(* CoDeSys 2.3 export: OSCAT311.TXT *)
(* Libraries: Standard.lib 4.10.05 11:14:46 *)

(* Global variable list: Constants *)
VAR_GLOBAL CONSTANT
	STRING_LENGTH : INT := 250;
	NETWORK_BUFFER_LONG_SIZE : UINT := 3999;
	NETWORK_BUFFER_SHORT_SIZE : UINT := 1459;
END_VAR




(* revisionhistory
hm 3. mar. 2007
	extended accuracy of pi2
	renamed T0 to Tk for better compatibility with other libraries
	renamed C t0 c0 for better compatibility

hm	2. may. 2007
	added RU universal gas constant

hm	1. oct. 2007
	added setup parameter STEP7

hm 31. oct. 2007
	added PN

hm	6. mar. 2008
	added setup Parameter EXTENDED_ASCII

hm	28. Mar. 2008
	added setup parameter STRING_LENGTH

hm	7. apr. 2008
	Deleted unused setup parameter Step7

hm	19. apr. 2008
	added setup parameter NETWORK_BUFFER_SIZE

hm	27. apr. 2008
	added PI05 and PI025

hm	18. may. 2008
	added charname lists
	renamed E to E1

hm	30. jun. 2008
	reduced size of string constants to 253 to avoid problems with target aixia DCUF

hm	21. sep. 2008
	added section language setup
	added section location setup

hm	20. oct. 2008
	changed to structured constants

hm	16. nov. 2008
	moved structured constants to global vars for compatibility reasons

hm	13. nov. 2009
	added network_buffer_short_size
	renamed network_buffer_long_size
	changed string length to 250
*)

(* Global variable list: Globale_Variablen *)
VAR_GLOBAL
	MATH : CONSTANTS_MATH;
	PHYS : CONSTANTS_PHYS;
	LANGUAGE : CONSTANTS_LANGUAGE;
	SETUP : CONSTANTS_SETUP;
	LOCATION : CONSTANTS_LOCATION;
END_VAR

(* Data type *)
TYPE CALENDAR :
STRUCT
	UTC : DT;						(* world time UTC *)
	LDT : DT;						(* local time *)
	LDATE : DATE;				(* local date *)
	LTOD : TOD;					(* local time of day *)
	YEAR : INT;					(* year of LDATE *)
	MONTH : INT;					(* month of LDATE *)
	DAY : INT;						(* day of LDATE *)
	WEEKDAY : INT;				(* weekday of LDATE *)
	OFFSET : INT;					(* Time Zone Offset for Local time in minutes *)
	DST_EN : BOOL;				(* daylight savings time enable *)
	DST_ON : BOOL;				(* true when daylight savings time os on *)
	NAME : STRING(5);			(* name of time zone *)
	LOCATION : INT;				(* location number pls see location setup *)
	LONGITUDE : REAL;			(* longitude of current location *)
	LATITUDE : REAL;			(* latitude of current location *)
	SUN_RISE : TOD;				(* sun_rise for current location *)
	SUN_SET : TOD;				(* sun_set for current location *)
	SUN_MIDDAY : TOD;			(* worldtime when sun stands at south position *)
	SUN_HEIGTH : REAL	;		(* suns heigth at midday, south position *)
	SUN_HOR : REAL;			(* sun angle horizontal 0 = north in degrees *)
	SUN_VER : REAL;			(* sun angle vertical above horizon in degrees *)
	NIGHT : BOOL;				(* true between sun_set and sun_rise *)
	HOLIDAY : BOOL;				(* true when holiday *)
	HOLY_NAME : STRING(30);	(* name of holiday *)
	WORK_WEEK : INT;			(* current work week *)
END_STRUCT
END_TYPE

(* revision history
hm	21. nov. 2008	rev 1.0
	original version

hm	8. feb. 2009	rev 1.1
	added sun position data

hm	10. mar. 2009	rev 1.2
	added work_week, sun_midday, sun_heigth
*)

(* Data type *)
TYPE COMPLEX :
STRUCT
	re : REAL;
	im : REAL;
END_STRUCT
END_TYPE


(* revision history
hm	18. oct. 2008
	original version

*)

(* Data type *)
TYPE CONSTANTS_LANGUAGE :
STRUCT
	(* Language Setup *)
	DEFAULT : INT := 1; (* 1=english, 2=german 3=french *)
	LMAX : INT := 3;
	WEEKDAYS : ARRAY[1..3, 1..7] OF STRING(10) :=	'Monday', 'Tuesday', 'Wednesday', 'Thursday', 'Friday', 'Saturday', 'Sunday',
													'Montag', 'Dienstag', 'Mittwoch', 'Donnerstag', 'Freitag', 'Samstag', 'Sonntag',
													'Lundi', 'Mardi', 'Mercredi', 'Jeudi', 'Vendredi', 'Samedi', 'Dimanche';
	WEEKDAYS2 : ARRAY[1..3, 1..7] OF STRING(2) :=	'Mo', 'Tu', 'We', 'Th', 'Fr', 'Sa', 'Su',
													'Mo', 'Di', 'Mi', 'Do', 'Fr', 'Sa', 'So',
													'Lu', 'Ma', 'Me', 'Je', 'Ve', 'Sa', 'Di';
	MONTHS : ARRAY[1..3, 1..12] OF STRING(10) :=	'January', 'February', 'March', 'April', 'May', 'June', 'July', 'August', 'September', 'October', 'November', 'December',
													'Januar', 'Februar', 'März', 'April', 'Mai', 'Juni', 'Juli', 'August', 'September', 'Oktober', 'November', 'Dezember',
													'Janvier', 'Février', 'mars', 'Avril', 'Mai', 'Juin', 'Juillet', 'Août', 'Septembre', 'Octobre', 'Novembre', 'Decembre';
	MONTHS3 : ARRAY[1..3, 1..12] OF STRING(3) :=	'Jan', 'Feb', 'Mar', 'Apr', 'May', 'Jun', 'Jul', 'Aug', 'Sep', 'Oct', 'Nov', 'Dec',
													'Jan', 'Feb', 'Mrz', 'Apr', 'Mai', 'Jun', 'Jul', 'Aug', 'Sep', 'Okt', 'Nov', 'Dez',
													'Jan', 'Fev', 'Mar', 'Avr', 'Mai', 'Jun', 'Jul', 'Aou', 'Sep', 'Oct', 'Nov', 'Dec';
	DIRS : ARRAY[1..3,0..15] OF STRING(3) :=		'N', 'NNE', 'NE', 'ENE', 'E', 'ESE', 'SE', 'SSE', 'S', 'SSW', 'SW', 'WSW', 'W', 'WNW', 'NW', 'NNW',
													'N', 'NNO', 'NO', 'ONO', 'O', 'OSO', 'SO', 'SSO', 'S', 'SSW', 'SW', 'WSW', 'W', 'WNW', 'NW', 'NNW',
													'N', 'NNO', 'NO', 'ONO', 'O', 'OSO', 'SO', 'SSO', 'S', 'SSW', 'SW', 'WSW', 'W', 'WNW', 'NW', 'NNW';
END_STRUCT
END_TYPE

(* revision history
hm	19. oct. 2008	rev 1.0
	original version

hm	22. oct. 2008	rev 1.1
	added directions DIRS

hm	23. dec. 2008	rev 1.2
	added french language

*)

(* Data type *)
TYPE CONSTANTS_LOCATION :
STRUCT
	(* location setup *)
	DEFAULT : INT := 1; (* 1=germany, 2=austria 3=france *)
	LMAX : INT := 3;

	(*	if month = 0 then F_day is the offset in days from easter
		used :0 = NOT used, 1 = used, -1..-7 menas the weekday before the specified DATE example -3 means wednesday before 23.11
	*)
	HOLIDAY : ARRAY[1..3, 0..29] OF HOLIDAY_DATA := (name := 'Neujahr', day := 1, month := 1, use := 1),
													(name := 'Heilig Drei Könige', day := 6, month := 1, use := 1),
													(name := 'Karfreitag', day := -2, month := 0, use := 1),
													(name := 'Ostersonntag', day := 0, month := 0, use := 1),
													(name := 'Ostermontag', day := 1, month := 0, use := 1),
													(name := 'Tag der Arbeit', day := 1, month := 5, use := 1),
													(name := 'Christi Himmelfahrt', day := 39, month := 0, use := 1),
													(name := 'Pfingstsonntag', day := 49, month := 0, use := 1),
													(name := 'Pfingstmontag', day := 50, month := 0, use := 1),
													(name := 'Fronleichnam', day := 60, month := 0, use := 1),
													(name := 'Augsburger Friedensfest', day := 8, month := 8, use := 0),
													(name := 'Maria Himmelfahrt', day := 15, month := 8, use := 1),
													(name := 'Tag der Deutschen Einheit', day := 3, month := 10, use := 1),
													(name := 'Reformationstag', day := 31, month := 10, use := 0),
													(name := 'Allerheiligen', day := 1, month := 11, use := 1),
													(name := 'Buss und Bettag', day := 23, month := 11, use := 0),
													(name := '1. Weihnachtstag', day := 25, month := 12, use := 1),
													(name := '2. Weihnachtstag', day := 26, month := 12, use := 1),
													(),
													(),
													(),
													(),
													(),
													(),
													(),
													(),
													(),
													(),
													(),
													(),
													(* the next 30 lines are for austrian holidays *)
													(name := 'Neujahr', day := 1, month := 1, use := 1),
													(name := 'Heilig Drei Könige', day := 6, month := 1, use := 1),
													(name := 'Karfreitag', day := -2, month := 0, use := 1),
													(name := 'Ostersonntag', day := 0, month := 0, use := 1),
													(name := 'Ostermontag', day := 1, month := 0, use := 1),
													(name := '', day := 1, month := 5, use := 0),
													(name := 'Christi Himmelfahrt', day := 39, month := 0, use := 1),
													(name := 'Pfingstsonntag', day := 49, month := 0, use := 1),
													(name := 'Pfingstmontag', day := 50, month := 0, use := 1),
													(name := 'Fronleichnam', day := 60, month := 0, use := 1),
													(name := '', day := 8, month := 8, use := 0),
													(name := 'Maria Himmelfahrt', day := 15, month := 8, use := 1),
													(name := '', day := 3, month := 10, use := 0),
													(name := '', day := 31, month := 10, use := 0),
													(name := 'Allerheiligen', day := 1, month := 11, use := 1),
													(name := 'Maria Empfängnis', day := 8, month := 12, use := 1),
													(name := '1. Weihnachtstag', day := 25, month := 12, use := 1),
													(name := '2. Weihnachtstag', day := 26, month := 12, use := 1),
													(),
													(),
													(),
													(),
													(),
													(),
													(),
													(),
													(),
													(),
													(),
													(),
													(* the next 30 lines are for french holidays *)
													(name := 'Nouvel an', day := 1, month := 1, use := 1),
													(name := 'St Valentin', day := 14, month := 2, use := 0),
													(name := 'Vendredi Saint (alsace)', day := -2, month := 0, use := 0),
													(name := 'Dimanche de pâques', day := 0, month := 0, use := 1),
													(name := 'Lundi de pâques', day := 1, month := 0, use := 1),
													(name := 'Jeudi de Ascension', day := 39, month := 0, use := 1),
													(name := 'dimanche de Pentecôte ', day := 49, month := 0, use := 1),
													(name := 'jeudi de la Trinité', day := 60, month := 0, use := 0),
													(name := 'Fête du travail', day := 1, month := 5, use := 1),
													(name := 'Victoire 1945 ', day := 8, month := 5, use := 1),
													(name := 'Prise de La bastille', day := 14, month := 7, use := 1),
													(name := '15 Août 1944', day := 15, month := 8, use := 1),
													(name := 'Halloween', day := 31, month := 10, use := 0),
													(name := 'Armistice 1918', day := 11, month := 11, use := 1),
													(name := 'Noël', day := 25, month := 12, use := 1),
													(name := 'Saint Étienne (alsace)', day := 26, month := 12, use := 0),
													(name := 'Fête de la musique', day := 21, month := 6, use := 0),
													(),
													(),
													(),
													(),
													(),
													(),
													(),
													(),
													(),
													(),
													(),
													(),
													();

END_STRUCT
END_TYPE


(* revision history
hm	20. oct. 2008	rev 1.0
	original version

hm	23. dec. 2008	rev 1.1
	added french holidays
*)

(* Data type *)
TYPE CONSTANTS_MATH :
STRUCT
	PI : REAL := 	3.14159265358979323846264338327950288;	(* Kreiszahl PI *)
	PI2 : REAL := 	6.28318530717958647692528676655900576;	(* PI * 2 *)
	PI4 : REAL :=  12.56637061435917295385057353311801152;	(* PI * 4 *)
	PI05 : REAL :=  1.5707963267949;						(* PI / 2 *)
	PI025 : REAL := 0.785398163397448;						(* PI / 4 *)
	PI_INV : REAL := 0.318309886183791;						(* 1 / PI *)
	E : REAL := 	2.71828182845904523536028747135266249;	(* Eulersche Konstante e *)
	E_INV : REAL := 0.367879441171442;						(* 1 / e *)
	SQ2 : REAL :=	1.4142135623731;						(* Wurzel von 2 *)
END_STRUCT
END_TYPE



(* revision history
hm	26.10.2008	rev 1.0
	original version

*)

(* Data type *)
TYPE CONSTANTS_PHYS :
STRUCT
	C : REAL := 299792458.0;				(* Lichtgeschwindigkeit in m/s *)
	E : REAL := 1.60217653E-19;				(* elementarladung in Colomb = A * s *)
	G : REAL := 9.80665; 						(* Erdbeschleunigung in m / s² *)
	T0 : REAL := -273.15;						(* absoluter Nullpunkt in °C *)
	RU : REAL := 8.314472; 					(* Universelle Gaskonstante in J / (mol · K) *)
	PN : REAL := 101325.0;					(* NormalDruck in Pa *)
END_STRUCT
END_TYPE



(* revision history
hm	18.10.2008	rev 1.0
	original version

hm	13. mar. 2009	rev 1.1
	real constants updated to new systax using dot

*)

(* Data type *)
TYPE CONSTANTS_SETUP :
STRUCT
	(* setup Parameters *)
	EXTENDED_ASCII : BOOL := TRUE;
	CHARNAMES : ARRAY[1..4] OF STRING(253) := ';"&quot;&&amp;<&lt;>&gt;€&euro; &nbsp;¡&iexcl;¢&cent;£&pound;¤&curren;¥&yen;¦&brvbar;§&sect;¨&uml;©&copy;ª&ordf;«&laquo;¬&not;­&shy;®&reg;¯&macr;°&deg;±&plusmn;²&sup2;³&sup3;´&acute;µ&micro;¶&para;·&middot;¸&cedil;¹&sup1;º&ordm;»&raquo;¼&frac14;Û&Ucirc;',
		';¾&frac34;¿&iquest;À&Agrave;Á&Aacute;Â&Acirc;Ã&Atilde;Ä&Auml;Å&Aring;Æ&AElig;Ç&Ccedil;È&Egrave;É&Eacute;Ê&Ecirc;Ë&Euml;Ì&Igrave;Í&Iacute;Î&Icirc;Ï&Iuml;Ð&ETH;Ñ&Ntilde;Ò&Ograve;Ó&Oacute;Ô&Ocirc;Õ&Otilde;Ö&Ouml;×&times;Ø&Oslash;Ù&Ugrave;Ú&Uacute;½&frac12;',
		';Ü&Uuml;Ý&Yacute;Þ&THORN;ß&szlig;à&agrave;á&aacute;â&acirc;ã&atilde;ä&auml;å&aring;æ&aelig;ç&ccedil;è&egrave;é&eacute;ê&ecirc;ë&euml;ì&igrave;í&iacute;î&icirc;ï&iuml;ð&eth;ñ&ntilde;ò&ograve;ó&oacute;ô&ocirc;õ&otilde;ö&ouml;÷&divide;ø&oslash;ù&ugrave;',
		';ú&uacute;û&ucirc;ü&uuml;ý&yacute;þ&thorn;ÿ&yuml;';
	MTH_OFS : ARRAY[1..12] OF INT := 0,31,59,90,120,151,181,212,243,273,304,334;
	DECADES : ARRAY[0..8] OF REAL := 1,10,100,1000,10000,10000,100000,1000000,10000000;
END_STRUCT
END_TYPE

(* revision history
hm	24.10.2008	rev 1.0
	original version

*)

(* Data type *)
TYPE ESR_DATA :
STRUCT
	TYP : BYTE;
	ADRESS : STRING(10);
	DS : DT;
	TS : TIME;
	DATA : ARRAY[0..7] OF BYTE;
END_STRUCT
END_TYPE


(* revision history
hm	18. oct. 2008
	original version

*)

(* Data type *)
TYPE HOLIDAY_DATA :
STRUCT
	NAME : STRING(30);
	DAY : SINT;
	MONTH : SINT;
	USE : SINT;
END_STRUCT
END_TYPE


(* revision history
hm	18. oct. 2008
	original version

*)

(* Data type *)
TYPE NETWORK_BUFFER :
STRUCT
	SIZE : UINT;
	BUFFER : NW_BUF_LONG;
END_STRUCT
END_TYPE


(* revision history
hm	18. oct. 2008
	original version

hm 13. nov. 2009
	use constant network_buffer_long_size

*)

(* Data type *)
TYPE NETWORK_BUFFER_SHORT :
STRUCT
	SIZE : UINT;
	BUFFER : NW_BUF_SHORT;
END_STRUCT
END_TYPE


(* revision history
hm 13. nov. 2009
	original version

*)

(* Data type *)
TYPE
	NW_BUF_LONG  : ARRAY[0..NETWORK_BUFFER_LONG_SIZE] OF BYTE;
END_TYPE

(* Data type *)
TYPE
	NW_BUF_SHORT : ARRAY[0..NETWORK_BUFFER_SHORT_SIZE] OF BYTE;
END_TYPE

(* Data type *)
TYPE REAL2 :
STRUCT
	R1 : REAL;	(* small value *)
	RX : REAL;	(* big value *)
END_STRUCT
END_TYPE


(* revision history
hm	18. oct. 2008
	original version

*)

(* Data type *)
TYPE SDT :
STRUCT
	YEAR : INT;
	MONTH : INT;
	DAY : INT;
	WEEKDAY : INT;
	HOUR : INT;
	MINUTE : INT;
	SECOND : INT;
	MS : INT;
END_STRUCT
END_TYPE


(* revision history
hm	18. oct. 2008
	original version

*)

(* Data type *)
TYPE TIMER_EVENT :
STRUCT
	TYP : BYTE;
	CHANNEL : BYTE;
	DAY : BYTE;
	START : TOD;
	DURATION : TIME;
	LAND : BYTE;
	LOR : BYTE;
	LAST : DWORD;
END_STRUCT
END_TYPE


(* revision history
hm	18. oct. 2008
	original version

*)

(* Data type *)
TYPE URL :
STRUCT
	PROTOCOL : STRING(10);
	USER : STRING(20);
	PASSWORD : STRING(20);
	DOMAIN : STRING(80);
	PORT : WORD;
	PATH : STRING(80);
	QUERY : STRING(40);
	ANCHOR : STRING(40);
END_STRUCT
END_TYPE


(* revision history
hm	18. oct. 2008
	original version

*)

(* Data type *)
TYPE VECTOR_3 :
STRUCT
	X : REAL;
	Y : REAL;
	Z : REAL;
END_STRUCT
END_TYPE


(* revision history
hm	18. oct. 2008
	original version

*)

(* POU PLC_PRG, CFC *)
PROGRAM PLC_PRG
VAR
END_VAR
_CFC_ (* Continuous Function Chart, elements in execution order *)
_END_CFC_
END_PROGRAM

(* POU Buffer Management/_BUFFER_CLEAR, ST *)
FUNCTION _BUFFER_CLEAR : BOOL
VAR_INPUT
	PT : POINTER TO BYTE;
	SIZE : UINT;
END_VAR
VAR
	ptw : POINTER TO DWORD;
	temp: DWORD;
	end, end32 : DWORD;
END_VAR


(*
version 1.2	31. oct. 2008
programmer 	hugo
tested by	oscat

this function will initialize a given array of byte with 0.
the function needs to be called:	_buffer_clear(adr("array"),sizeof("array"));
this function will manipulate a given array.
the function manipulates the original array, it rerturnes true when finished.
because this function works with pointers its very time efficient and it needs no extra memory.

*)
(* this routine uses 32 bit access to gain speed *)
(* first access bytes till pointer is aligned for 32 bit access *)
temp := pt;
end := temp + UINT_TO_DWORD(size);
end32 := end - 3;
WHILE (pt < end) AND ((temp AND 16#00000003) > 0) DO
	pt^ := 0;
	pt := pt + 1;
	temp := temp + 1;
END_WHILE;
(* pointer is aligned, now copy 32 bits at a time *)
ptw := pt;
WHILE ptw < end32 DO (* *)
	ptw^ := 0;
	ptw := ptw + 4;
END_WHILE;
(* copy the remaining bytes in byte mode *)
pt := ptw;
WHILE pt < end DO
	pt^ := 0;
	pt := pt + 1;
END_WHILE;

_BUFFER_CLEAR := TRUE;

(* revision History
hm 	5. mar. 2008	rev 1.0
	original version

hm	16. mar. 2008	rev 1.1
	added type conversion to avoid warnings under codesys 30
	chaged type of input size to uint
	deleted unused variable i

hm	31. oct. 2008	rev 1.2
	corrected an error while routine would write outside of arrays

*)
END_FUNCTION

(* POU Buffer Management/_BUFFER_INIT, ST *)
FUNCTION _BUFFER_INIT : BOOL
VAR_INPUT
	PT : POINTER TO BYTE;
	SIZE : UINT;
	INIT : BYTE;
END_VAR
VAR
	ptw : POINTER TO DWORD;
	temp : DWORD;
	end, end32 : DWORD;
END_VAR


(*
version 1.2	31. oct. 2008
programmer 	hugo
tested by	oscat

this function will initialize a given array of byte with init.
the function needs to be called:	_buffer_init(adr("array"),sizeof("array"),init);
this function will manipulate a given array.
the function manipulates the original array, it rerturnes true when finished.
because this function works with pointers its very time efficient and it needs no extra memory.

*)
(* this routine uses 32 bit access to gain speed *)
(* first access bytes till pointer is aligned for 32 bit access *)
temp := pt;
end := temp + UINT_TO_DWORD(size);
end32 := end - 3;
WHILE (pt < end) AND ((temp AND 16#00000003) > 0) DO
	pt^ := init;
	pt := pt + 1;
	temp := temp + 1;
END_WHILE;
(* pointer is aligned, now copy 32 bits at a time *)
ptw := pt;
temp := SHL(BYTE_TO_DWORD(init),24) OR SHL(BYTE_TO_DWORD(init),16) OR SHL(BYTE_TO_DWORD(init),8) OR BYTE_TO_DWORD(init);
WHILE ptw < end32 DO
	ptw^ := temp;
	ptw := ptw + 4;
END_WHILE;
(* copy the remaining bytes in byte mode *)
pt := ptw;
WHILE pt < end DO
	pt^ := init;
	pt := pt + 1;
END_WHILE;

_BUFFER_INIT := TRUE;

(* revision History
hm 	5. mar. 2008	rev 1.0
	original version

hm	16. mar. 2008	rev 1.1
	added type conversion to avoid warnings under codesys 3.0
	chaged type of input size to uint.

hm	31. oct. 2008	rev 1.2
	corrected an error while routine would write outside of arrays

*)
END_FUNCTION

(* POU Buffer Management/_BUFFER_INSERT, ST *)
FUNCTION _BUFFER_INSERT : BOOL
VAR_INPUT
	STR : STRING(STRING_LENGTH);
	POS : INT;
	PT : POINTER TO ARRAY[0..32767] OF BYTE;
	SIZE : UINT;
END_VAR
VAR
	end : INT;
	lx: INT;
	i: INT;
END_VAR


(*
version 1.4	12. nov. 2009
programmer 	hugo
tested by		oscat

this function will initialize a given array of byte with init.
the function needs to be called:	_buffer_init(adr("array"),sizeof("array"),init);
this function will manipulate a given array.
the function manipulates the original array, it rerturnes true when finished.
because this function works with pointers its very time efficient and it needs no extra memory.

*)
lx := LEN(str);
end := pos + lx;
(* first move the upper part of the buffer to make space for the string *)
FOR i := UINT_TO_INT(size) - 1 TO end BY -1 DO
	pt^[i] := pt^[i-lx];
END_FOR;
(* copy the string *)
_BUFFER_INSERT := _STRING_TO_BUFFER(str, pos, PT, size);


(* revision History
hm 	9. mar. 2008	rev 1.0
	original version

hm	16. mar. 2008	rev 1.1
	changed type of input size to uint

hm	13. may. 2008	rev 1.2
	changed type of pointer to array[1..32767]
	changed size of string to STRING_LENGTH

hm	23. mar. 2009	rev 1.3
	avoid writing to input pos

hm	12. nov. 2009	rev 1.4
	code optimized

*)
END_FUNCTION

(* POU Buffer Management/_STRING_TO_BUFFER, ST *)
FUNCTION _STRING_TO_BUFFER : BOOL
VAR_INPUT
	STR : STRING(STRING_LENGTH);
	POS : INT;
	PT : POINTER TO ARRAY[0..32767] OF BYTE;
	SIZE : UINT;
END_VAR
VAR
	ps : POINTER TO BYTE;
	i: INT;
	end: INT;
END_VAR


(*
version 1.3	12. nov. 2009
programmer 	hugo
tested by		oscat

this function will copy a string into an array of byte starting at position pos.
the function needs to be called:	_String_To_buffer(str, pos, adr("array"),sizeof("array"));
this function will manipulate the array directly in memory and returns true when finished.
because this function works with pointers its very time efficient and it needs no extra memory.

*)
ps := ADR(str);
end := MIN(pos + LEN(str), UINT_TO_INT(size));
IF end > 0 THEN end := end -1; END_IF;
FOR i := pos TO end DO
	pt^[i] := ps^;
	ps := ps + 1;
END_FOR;

_STRING_TO_BUFFER := TRUE;

(* revision History

hm 	5. mar. 2008	rev 1.0
	original version

hm	16. mar. 2008	rev 1.1
	changed type of input size to uint

hm	13. may. 2008	rev 1.2
	changed type of pointer to array[1..32767]
	changed size of string to STRING_LENGTH

hm	12. nov. 2009	rev 1.3
	limit end to size - 1

*)
END_FUNCTION

(* POU Buffer Management/BUFFER_COMP, ST *)
FUNCTION BUFFER_COMP : INT
VAR_INPUT
	PT1 : POINTER TO ARRAY[0..32767] OF BYTE;
	SIZE1 : INT;
	PT2 : POINTER TO ARRAY[0..32767] OF BYTE;
	SIZE2 : INT;
	START : INT;
END_VAR
VAR
	i, j, end : INT;
	firstbyte: BYTE;
END_VAR

(*
version 1.1	12. nov. 2009
programmer 	hugo
tested by	oscat


 
*)
(* search for first character match *)
IF size2 <= size1 THEN
	end := size1 - size2;
	firstbyte := PT2^[0];
	FOR i := START TO end DO
		IF PT1^[i] = firstbyte THEN
			(* first character matches, now compare rest of array *)
			j := 1;
			WHILE j < size2 DO
				IF pt2^[j] <> pt1^[j+i] THEN EXIT; END_IF;
				j := j + 1;
			END_WHILE;
			(* when J > size2 a match was found return the position i in buffer1 *)
			IF j = size2 THEN
				BUFFER_COMP := i;
				RETURN;
			END_IF;
		END_IF;
	END_FOR;
END_IF;
BUFFER_COMP := -1;


(*
hm 14. nov. 2008	rev 1.0
	original version

hm	12. nov. 2009	rev 1.1
	performance increase

*)
END_FUNCTION

(* POU Buffer Management/BUFFER_SEARCH, ST *)
FUNCTION BUFFER_SEARCH : INT
VAR_INPUT
	PT : POINTER TO ARRAY[0..32767] OF BYTE;
	SIZE : UINT;
	STR : STRING(STRING_LENGTH);
	POS : UINT;
	IGN : BYTE;
END_VAR
VAR
	ps : POINTER TO ARRAY[0..255] OF BYTE;
	i: INT;
	end: INT;
	k: INT;
	lx: INT;
END_VAR


(*
version 1.3	12. nov. 2009
programmer 	hugo
tested by	oscat

this function will search for a string STR in an array of byte starting at position pos.
the function needs to be called:	buffer_search(adr("array"),sizeof("array"), STR, POS, IGN);
because this function works with pointers its very time efficient and it needs no extra memory.
The function returns the position of the first character of the string in the array if found.
a 0 is returned if the string is not found in the array.
The parameter IGN specifies a wildcard character in the search string.

*)
ps := ADR(str);
lx := LEN(str);
end := MIN(UINT_TO_INT(size) - lx, UINT_TO_INT(size - 1));
lx := lx - 1;
FOR i := UINT_TO_INT(pos) TO end DO
	FOR k := 0 TO lx DO
		IF (ps^[k] <> ign) AND (ps^[k] <> pt^[i+k]) THEN EXIT; END_IF;
	END_FOR;
	IF k > lx THEN
		BUFFER_SEARCH := i;
		RETURN;
	END_IF;
END_FOR;
BUFFER_SEARCH := 0;


(* revision History

hm 5. mar. 2008	rev 1.0
	original version

hm	16. mar. 2008	rev 1.1
	chaged type of input size to uint

hm	13. may. 2008	rev 1.2
	changed type of pointer to array[1..32767]
	changed size of string to STRING_LENGTH

hm	12. nov. 2009	rev 1.3
	limit end to array size

*)
END_FUNCTION

(* POU Buffer Management/BUFFER_TO_STRING, ST *)
FUNCTION BUFFER_TO_STRING : STRING(STRING_LENGTH)
VAR_INPUT
	PT : POINTER TO ARRAY[0..32767] OF BYTE;
	SIZE : UINT;
	START : UINT;
	STOP : UINT;
END_VAR
VAR
	ps : POINTER TO BYTE;
	i : UINT;
	stp: UINT;
	sta: UINT;
END_VAR


(*
version 1.5	12. nov. 2009
programmer 	hugo
tested by		oscat

this function will retrieve a string from an array of byte starting at position start and stop at position stop.
the function needs to be called:	buffer_TO_String(adr("array"),sizeof("array"), start, stop);
because this function works with pointers its very time efficient and it needs no extra memory.

*)
ps := ADR(BUFFER_TO_STRING);
IF size = 0 THEN RETURN; END_IF;
sta := MIN(start, size -1);
stp := MIN(stop, size -1);

(* check for maximum string_length *)
IF UINT_TO_INT(stp - sta + 1) >= STRING_LENGTH THEN
	stp := sta + INT_TO_UINT(STRING_LENGTH) - 1;
END_IF;

FOR i := sta TO stp DO
	ps^ := pt^[i];
	ps := ps + 1;
END_FOR;

(* terminate the string *)

ps^ := 0;



(* revision History
hm 	5. mar. 2008	rev 1.0
	original version

hm	16. mar. 2008	rev 1.1
	changed type of input size to uint

hm	13. may. 2008	rev 1.2
	changed type of pointer to array[0..32767]
	changed size of string to STRING_LENGTH

hm	12. jun. 2008	rev 1.3
	check for pointer overrun
	change input start and stop to uint
	added type conversions to avoid warnings under codesys 3.0

hm	23. mar. 2009	rev 1.4
	avoid writing to input stop

hm	12. nov. 2009 rev 1.5
	limit start and stop to size -1

*)
END_FUNCTION

(* POU Building/actuators/ACTUATOR_2P, ST *)
FUNCTION_BLOCK ACTUATOR_2P
VAR_INPUT
	IN : BYTE;
	TEST : BOOL;
	ARE : BOOL := TRUE;
END_VAR
VAR_IN_OUT
	ARX : BOOL;
END_VAR
VAR_INPUT CONSTANT
	CYCLE_TIME : TIME;
	SENS : BYTE;
	SELF_ACT_TIME : TIME;
	SELF_ACT_PULSE : TIME;
	SELF_ACT_CYCLES : INT := 1;
END_VAR
VAR_OUTPUT
	OUT : BOOL;
	ARO : BOOL;
END_VAR
VAR
	timer : AUTORUN;
	pwgen : GEN_PULSE;
END_VAR


(*
version 2.1	24. jan. 2009
programmer 	hugo
tested by		oscat

this is an intelligent actuator interface for any 2point actuator like coil drive.
the 2Point actuator can only switch on/off and therefore the input must be converted to on/off cycles.
the interface can be programmed with double click on the symbol.
in addition a self_act_time and self_act_cycles ca be programmed to switch n times on/off every self_act_time to avoid a valve to freeze.
the input value must be between 0 and 255. with the setup variable sens one can specify what must be the minimum input to turn the valve on at all.
at the same time an input > 255-sens will turn the valve on at all times.


*)
(* run the autorun timer *)
timer(trun := SELF_ACT_PULSE * (2 * SELF_ACT_CYCLES), toff := SELF_ACT_TIME, Test := TEST, ARE := ARE, arx := ARX);
ARO := timer.ARO;

(* run the pulse width generator *)
IF aro THEN
	pwgen(PTL := SELF_ACT_PULSE, PTH := SELF_ACT_PULSE);
	out := pwgen.Q;
ELSIF in < sens THEN
	out := FALSE;
ELSIF in > BYTE#255 - sens THEN
	out := TRUE;
ELSE
	pwgen.PTH := (CYCLE_TIME * BAND_B(IN,SENS)) / 255;
	pwgen.PTL := CYCLE_TIME - pwgen.PTH;
	pwgen();
	out := pwgen.Q;
END_IF;



(* revision history
hm	7.10.2006 		rev 1.1
	changed error pos could not reach 1 or 0 under certain conditions due to error in code.
	changed on and off in force and force_in for better usability.

hm	17.1.2007		rev 1.2
	deleted unused variable time_overflow

hm	15.9.2007		rev 1.3
	replaced time() with T_PLC_MS for compatibility and performance reasons

hm	19. 11 2007		rev 1.4
	replaced left over statement time() with tx

hm	27. 12. 2007	REV 1.5
	CHANGED CODE FOR BETTER PERFORMANCE

hm	21. oct. 2008	rev 1.6
	code optimized

hm	23. nov. 2008	rev 2.0
	new code using library modules

hm	24. jan. 2009	rev 2.1
	deleted unused var inb
*)
END_FUNCTION_BLOCK

(* POU Engineering/measurements/CYCLE_TIME, ST *)
FUNCTION_BLOCK CYCLE_TIME
VAR_INPUT
	RST : BOOL;
END_VAR
VAR_OUTPUT
	ct_min : TIME;
	ct_max : TIME;
	ct_last : TIME;
	systime : TIME;
	sysdays : INT;
	cycles : DWORD;
END_VAR
VAR
	last_cycle : TIME;
	tx: TIME;
	init: BOOL;
END_VAR


(*
	version 1.2	16 sep 2007
	programmer 	hugo
	tested BY		hans

this function block measures the cycle time and displays the last, min and max cycle time of the current task.
the resolution is 1ms.
the cycles output is a dword counter which counts the cycles.
a rst pulse on the input will reset all data.


*)
tx := DWORD_TO_TIME(T_PLC_MS()) - last_cycle;
IF rst THEN
	ct_min := t#10h;
	ct_max := t#0ms;
	cycles := 0;
ELSIF last_cycle > t#0s THEN
	IF tx < ct_min THEN ct_min := tx;
	ELSIF tx > ct_max THEN ct_max := tx;
	END_IF;
	ct_last := tx;
ELSIF ct_min = t#0s THEN
	ct_min := t#0s - t#1ms;
END_IF;
IF init THEN
	systime := systime + tx;
		IF systime >= t#1d THEN
			systime := systime - t#1d;
			sysdays := sysdays + 1;
		END_IF;
END_IF;
init := TRUE;
last_cycle := last_cycle + tx;
cycles := cycles + 1;

(*	revision history
hm 12.12.2006		rev 1.1
	added cycles output, a dword cycle counter.
hm 10.3.2007			rev 1.2
	changed initialization of ct_min to t#10h for compatibility with siemens s7

hm	16.9.2007		rev 1.2
	changed Time() in T_PLC_MS() for compatibility resons

*)
END_FUNCTION_BLOCK

(* POU Engineering/measurements/T_PLC_MS, ST *)
FUNCTION T_PLC_MS : DWORD
VAR CONSTANT
	debug : BOOL := 0;
	N : INT := 0;
	offset : DWORD := 0;
END_VAR
VAR
	tx : TIME;
END_VAR

(*
version 1.2	16. nov 2008
programmer 	hugo
tested by	oscat

T_PLC_MS reads the internal PLC timer and return the time, it has the advantage to be able to set a debug mode 
and speed up the counter to test the plc timer overrun which occurs every 50 days respectively 25 days at siemens S7
this routine also allows to correct the behavior of s7 where the internal plc counter will not count all 32 bits.

*)
tx := TIME();
T_PLC_MS := TIME_TO_DWORD(Tx);
(* hier muss die korrektur für step7 stattfinden
plctime muss den vollen wertebereich von time ausnutzen:
wenn bei step7 time -24tage bis plus 24 tage ist dann muss der timer auch beim überlauf auf -24tage springen 
und auf keinen fall auf 0 !!!!
für siemens muss ein weiterer fb im main eingebunden werden der sicherstellt das alle 32 bits durchgezählt werden.
es kann nur ein fb sein den er muss sich das oberste (32te) bit merken.
oder etwa spring s7 bei überlauf auf -24 tage????? dann wäre keine korrektur nötig.
*)
IF debug THEN
	T_PLC_MS := (SHL(T_PLC_MS,N) OR SHL(DWORD#1,N)-1) + OFFSET;
END_IF;

(* revision history
hm	14.9.2007	rev 1.0
	original version

hm	12. nov 2007	rev 1.1
	added temporaray variable tx because some compilers could not handle time() as an argument

hm	16. nov. 2008	rev 1.2
	initialized constants with 0 for compatibility reasons
*)
END_FUNCTION

(* POU Engineering/signal processing/OFFSET, ST *)
FUNCTION OFFSET : REAL
VAR_INPUT
	X : REAL;
	O1, O2, O3, O4 : BOOL;
	D : BOOL;
END_VAR
VAR_INPUT CONSTANT
	Offset_1 : REAL;
	Offset_2 : REAL;
	Offset_3 : REAL;
	Offset_4 : REAL;
	default : REAL;
END_VAR

(*
version 1.0	12 jan 2007
programmer 	oscat
tested by	oscat

The Function offset adds offsets to an analog signal depending on digital inputs.
all selected offsets are added at the same time.
with the input D a default value instead of the input X can be used.

*) 
IF D THEN OFFSET := default; ELSE OFFSET := X; END_IF;
IF O1 THEN OFFSET := OFFSET + offset_1; END_IF;
IF O2 THEN OFFSET := OFFSET + offset_2; END_IF;
IF O3 THEN OFFSET := OFFSET + offset_3; END_IF;
IF O4 THEN OFFSET := OFFSET + offset_4; END_IF;



(* revision history
hm	12. jan 2007
	original version


*)
END_FUNCTION

(* POU Building/actuators/AUTORUN, ST *)
FUNCTION_BLOCK AUTORUN
VAR_INPUT
	IN : BOOL;
	TEST : BOOL;
	ARE : BOOL := TRUE;
END_VAR
VAR_IN_OUT
	ARX : BOOL;
END_VAR
VAR_INPUT CONSTANT
	TRUN : TIME;
	TOFF : TIME;
END_VAR
VAR_OUTPUT
	OUT : BOOL;
	ARO : BOOL;
END_VAR
VAR
	timer : _RMP_B;
	val : BYTE;
END_VAR



(*
version 1.0	20. nov 2008
programmer 	hugo
tested by	oscat




*)
(* run the integrator when T_off > T#0s *)
IF TOFF > T#0s THEN
	timer(DIR:= OUT, TR := SEL(OUT, TOFF, TRUN), RMP := val);
ELSE
	val := 255;
END_IF;


(* when timer = 0 or test then initiate autorun until timer reaches 255 *)
IF (NOT ARX AND ARE AND val = 0) OR TEST THEN
	val := 0;
	ARO := TRUE;
	ARX := TRUE;
ELSIF val = 255 AND ARO THEN
	ARO := FALSE;
	ARX := FALSE;
END_IF;

(* output is true when autorun ARO is true or in = TRUE *)
out := IN OR ARO;



(* revision history
hm 20. nov. 2008	rev 1.0
	original version

*)
END_FUNCTION_BLOCK

(* POU Engineering/signal generators/_RMP_B, ST *)
FUNCTION_BLOCK _RMP_B
VAR_INPUT
	DIR : BOOL;  (* true = up *)
	E : BOOL := TRUE;
	TR : TIME;
END_VAR
VAR_IN_OUT
	RMP : BYTE;
END_VAR
VAR
	tx, tl : DWORD;
	step : INT;
	init: BOOL;
	last_dir: BOOL;
END_VAR


(*
version 1.1	20. nov. 2008
programmer 	hugo
tested by	oscat


_RMP_B generates a ramp on an external var of type byte
tr is the total ramp time, E is an enable and dir the direction of the ramp

*)
tx := T_PLC_MS();
IF E AND init THEN
	(* we need to set tl = tx when direction changes *)
	IF dir XOR last_dir THEN
	 tl := tx;
	 last_dir := dir;
	END_IF;
	(* check_elapsed time and calculate only if necessary *)
	IF tr > t#0s THEN
		step := DWORD_TO_INT(SHL(tx-tl, 8) / TIME_TO_DWORD(TR));
	ELSE
		step := 255;
	END_IF;
	IF step > 0 THEN
		(* perform the step on the ramp *)
		tl := tx;
		(* calculate the step response *)
		IF NOT dir THEN step := - step; END_IF;
		rmp := INT_TO_BYTE(LIMIT(0, BYTE_TO_INT(rmp) + step, 255));
	END_IF;
ELSE
	tl := tx;
	init := TRUE;
END_IF;


(* revison history
hm	22. oct. 2008	rev 1.0
	original version

hm	20. nov. 2008	rev 1.1
	set default for E to be TRUE
	added init

*)
END_FUNCTION_BLOCK

(* POU Engineering/signal generators/GEN_PULSE, ST *)
FUNCTION_BLOCK GEN_PULSE
VAR_INPUT
	ENQ : BOOL := TRUE;
	PTH : TIME;
	PTL : TIME;
END_VAR
VAR_OUTPUT
	Q : BOOL;
END_VAR
VAR
	tx: TIME;
	tn: TIME;
	init: BOOL;
END_VAR

(*
version 1.3	13. nov. 2009
programmer 	hugo
tested by		oscat

GEN_PULSE uses the internal sps timer to generate a continuous output waveform with programmable high and low time.
the accuracy of gen_pulse is depending on the system timer.
when time is 0 the high and low times are exactly one cycle.
ENQ = TRUE will start and ENQ = FALSE will stop the generator.

*)
(* read system timer *)
IF enq THEN
	tx := DWORD_TO_TIME(T_PLC_MS());
	IF NOT init THEN init := TRUE; tn := tx; END_IF;
	IF tx >= tn THEN
		Q := NOT Q;
		tn := tn + SEL(Q,PTL,PTH);
	END_IF;
ELSE
	Q := FALSE;
	init := FALSE;
END_IF;



(* revision history
hm	29. jun. 2008	rev 1.0
	original version

hm	23. nov. 2008	rev 1.1
	set default for enq to be true

hm	18. jul. 2009	rev 1.2
	improved performance

hm	13. nov. 2009	rev 1.3
	corrected error

*)
END_FUNCTION_BLOCK

(* POU Engineering/control/BAND_B, ST *)
FUNCTION BAND_B : BYTE
VAR_INPUT
	X : BYTE;
	B : BYTE;
END_VAR



(*
version 1.0	21. Nov. 2008
programmer 	hugo
tested by	oscat

BAND_B will limit X to B <= X <= 255-B. while X < B the resulkt will be 0 and while X > 255-B the output will be 255
otherwise the result = X.

*)
IF X < B THEN
	BAND_B := 0;
ELSIF X > BYTE#255-B THEN
	BAND_B := 255;
ELSE
	BAND_B := X;
END_IF;



(* revision history
hm	21. nov. 2008	rev 1.0
	original version

*)
END_FUNCTION

(* POU Building/actuators/ACTUATOR_3P, ST *)
FUNCTION_BLOCK ACTUATOR_3P
VAR_INPUT
	in : REAL;
	force : BOOL;
	on : BOOL;
	end_pos : BOOL;
	diag : BOOL;
END_VAR
VAR_INPUT CONSTANT
	min_ontime : TIME := t#10s;
	min_offtime : TIME := t#10s;
	max_runtime : TIME := t#60s;
	auto_diag_time : TIME := t#10d;
	cal_runtime : TIME := t#600s;
	switch_available: BOOL;
END_VAR
VAR_OUTPUT
	out1 : BOOL;
	out2 : BOOL;
	pos : REAL;
	busy : BOOL;
	error : BOOL;
END_VAR
VAR
	val: REAL;
	tx : TIME;
	last_diag: TIME;
	last : TIME;
	runtime_1 : TIME;
	runtime_2 : TIME;
	state : INT;
	rout: FT_RMP;
	end : R_TRIG;
	cal_timer: TIME;
	Tn: TIME;
END_VAR


(*
version 1.3	 15 sep 2007
programmer 	hugo
tested by	oscat

actuator_3P is an interface for a 3 point actuator.
a 3P actuator is a motor with 2 directions that drives a valve or flap. the position of the valve or flap is controlled by runtime of the motor foreward or backward.
the available inputs are:
in is a real value which specifies the position of the actuator, 0 = 0% and 1 = 100% any value <0 or > 1 is limited to 0 or 1.
a force input must be low for normal operation and if switched high, the motor can only be controlled for 0% or 100% positions with the on input.
an and pos input is available for a end_pos switch, this switch indicates the valve or flap to be at either 0% or 100%
a diag input can at any time start a diag cycle which turns the motor towards the 0% position, then measures the runtime to 100% and then the runtime to 0%
these runtimes are stored and used for absolute positioning of the motor during normal operation.
a setup constand "auto_diag_time can be used to specify how often the actuator repeates this auto_diag cycla automatically.
at power on a cycle is perfomed automatically.
a 0 for this value means auto diag is never performed.

the outputs ar out1 and out2 for up and down direction of the motor. to avoid flickering the output can be programmed for min_ontime and min_offtime.
a pos outout indicates the absulute position of the actuator during operation and a busy output indicates the actuator is busy.
a error output is initiated when the specified max_runtime is reached by any direction during debug.
also when the up and down direction differs by more then 10% the error output is set.

for absolute positioning accuracy the actuator has a setup variable "cal_runtime" if this is set the actuator measures the total runtime of the motors and when this 
cal_runtime is exceeded it resets the actuator to 0% position and sets the output again to assure absolute accuracy.

autodiag and calibration can be shut off by setting the appropriate values to 0.
a switch_available setup variable specifies if end_pos switches are available.

*)
(* setup *)
Tn := DWORD_TO_TIME(T_PLC_MS());
tx := Tn - last;
end(clk := end_pos);

(* init only when first started *)
IF state = 0 THEN
	runtime_1 := max_runtime;
	runtime_2 := max_runtime;
	state := 1;
	rout(KR := 1000 / TIME_TO_REAL(runtime_1), KF := 1000 / TIME_TO_REAL(runtime_1) );
	tx := t#0s;
	last := Tn;
	last_diag := last;
END_IF;

(* check for end_sw and stop if reached *)
IF switch_available AND out1 AND end.Q THEN
	(* upper limit has been reached *)
	out1 := 0;
	rout(rmp := 0, in := 1);
	rout.Rmp := 1;
ELSIF switch_available AND out2 AND end.Q THEN
	(* lower limit has been reached *)
	out2 := 0;
	rout(rmp := 0, in := 0);
	rout.Rmp := 1;
END_IF;

(* check for min_offtime and min_ontime and return if it has not elapsed *)
IF NOT busy AND tx < min_offtime THEN
	RETURN;
ELSIF busy AND tx < min_ontime THEN
	RETURN;

(* check for last diag cycle and start diag if auto_diag_time has elapsed *)
ELSIF (tn - last_diag > auto_diag_time AND state > 10 AND auto_diag_time > t#0s) OR (diag AND state >= 10) THEN state := 1;

(* check if force pin is high *)
ELSIF force THEN state := 10;

(* check if calibration is necessary *)
ELSIF cal_timer > cal_runtime AND state = 99 AND cal_runtime > t#0s THEN state := 20;
END_IF;

(* state machine for operation *)
CASE state OF

1 :	(* diagnostic start *)
	(* all data is reset and out2 is turned on to make sure we start from top position *)
	last_diag := tn;
	diag := 0;
	state := 2;
	pos := 0;
	busy := 1;
	last := tn;
	out1 := 0;
	out2 := 1;
	RETURN;

2:	(* wait for max_runtime or end_pos to be reached *)
	IF tx < max_runtime AND NOT end.Q THEN RETURN; END_IF;
	state := 3;
	last := tn;
	out1 := 1;
	out2 := 0;
	RETURN;

3: 	(* measure runtime_2 *)
	IF tx < max_runtime AND NOT end.Q THEN RETURN; END_IF;
	state := 4;
	runtime_1 := tx;
	last := tn;
	out1 := 0;
	out2 := 1;
	RETURN;

4:	(* measure runtime_1 *)
	IF tx < max_runtime AND NOT end.Q THEN RETURN; END_IF;
	state := 99;
	runtime_2 := tx;
	last := tn;
	out2 := 0;
	busy := 0;
	(* reset the output ramp generator to the 0% position as the valve is after diags *)
	rout(rmp := 0, in := 0);
	rout.Rmp := 1;
	cal_timer := t#0s;
	IF DIFFER(TIME_TO_REAL(runtime_1), TIME_TO_REAL(runtime_2), TIME_TO_REAL(max_runtime) * 0.1) THEN error := TRUE;
	ELSIF runtime_1 > MULTIME(max_runtime, 0.9) AND switch_available THEN error := TRUE;
	ELSIF runtime_2 > MULTIME(max_runtime, 0.9) AND switch_available THEN error := TRUE;
	END_IF;
	RETURN;

10: (* force pin is active, outputs are forced on or off by the on pin *)
	IF on AND NOT out2 THEN val := 1;
	ELSIF NOT on AND NOT out1 THEN val := 0;
	END_IF;
	IF NOT force THEN state := 99; END_IF;

20 : (* calibrate to allow for correction of positioning error addig up *)
	cal_timer := t#0s;
	state := 21;
	pos := 0;
	busy := 1;
	last := tn;
	out1 := 0;
	out2 := 1;
	RETURN;

21:	(* after end_sw or max_runtime we can be sure to have reached the 0% position *)
	IF tx < max_runtime AND NOT end.Q THEN RETURN; END_IF;
	state := 99;
	out2 := 0;
	busy := 0;
	last := tn;
	rout(rmp := 0, in := 0);
	rout.Rmp := 1;
	RETURN;

99: (* normal operation *)
	(* only if input changes for an equivalent of min_ontime then change the output *)
	(* if there is a directional change then wait until last step is finished *)
	IF in < TIME_TO_REAL(min_ontime)/TIME_TO_REAL(max_runtime)/2 THEN val := 0;
	ELSIF in > 1 - TIME_TO_REAL(min_ontime)/TIME_TO_REAL(max_runtime)/2 THEN val := 1;
	ELSIF differ(LIMIT(0,in,1), val, TIME_TO_REAL(min_ontime) / TIME_TO_REAL(max_runtime)) OR in = 0 OR in = 1 THEN
		IF in < val AND NOT out1 THEN val := in;
		ELSIF in > val AND NOT out2 THEN val := in;
		END_IF;
	END_IF;

END_CASE;

(* output ramp generator *)
rout(in := val);
out1 := rout.busy AND rout.UD;
out2 := rout.busy AND NOT rout.UD;
pos := rout.out;

(* set the busy output and if busy goes low, then set the last time in order to check for min_offtime *)
IF NOT busy AND rout.busy THEN
	last := tn;
ELSIF busy AND NOT rout.busy THEN
	cal_timer := cal_timer + tx;
	last := tn;
END_IF;
busy := rout.busy;



(* revision history

19.10.2006	rev 1.1
	added security checks for end_switch to avoid overrun of the end_switch, hans

23.1.2007		rev 1.2
	deleted unused variables force_on and force_off

15.9.2007	hm	rev 1.3
	replaced Time() with T_PLC_MS for compatibility and performance reasons

*)
END_FUNCTION_BLOCK

(* POU Mathematical/functions/FT_RMP, ST *)
FUNCTION_BLOCK FT_RMP
VAR_INPUT
	Rmp : BOOL := TRUE;
	in : REAL;
	KR : REAL;
	KF : REAL;
END_VAR
VAR_OUTPUT
	out : REAL;
	busy : BOOL;
	UD : BOOL;
END_VAR
VAR
	tx: TIME;
	last: TIME;
	init: BOOL;
END_VAR

(*
	version 1.4	25 jan 2008
	programmer 	oscat
	tested BY		oscat

this ramp function follows an input signal with a linear ramp up or down, the up or down speed can be set with KF and KR.
a K factor of 1 means 1 unit per second on the output. K factors can only be positive and not negative.
a busy output signals the ramp is running or busy false means the in value is present on the output.
a rmp input false means the output follows the input dierctly while a rmp = true means the output follows the input with a ramp.
a updn output signal the directon of the ramp (up or down).

*)
(* read system time *)
tx := DWORD_TO_TIME(T_PLC_MS()) - last;

IF NOT init THEN
	init := TRUE;
	last := tx;
	tx := t#0s;
	out := in;
END_IF;
IF NOT rmp THEN
	out := in;
	busy := FALSE;
ELSIF out > in THEN
	(* ramp down *)
	out := out - TIME_TO_REAL(tx) * 0.001 * KF;
	out := MAX(in, out);
ELSIF out < in THEN
	(* ramp up *)
	out := out + TIME_TO_REAL(tx) * 0.001 * KR;
	out := MIN(in, out);
END_IF;

(* set busy and dir flags *)
IF out < in THEN
	busy := TRUE;
	ud := TRUE;
ELSIF out > in THEN
	busy := TRUE;
	ud := FALSE;
ELSE
	busy := FALSE;
END_IF;
last := last + tx;


(* revision history:

hm 8.10.2006			rev 1.1
	added ud output

hm 12. feb 2007		rev 1.2
	added init variable and corrected a possible startup problem

hm	17. sep 2007	rev 1.3
	replaced time() with t_plc_ms() for compatibility reasons

hm	25. jan 2008	rev 1.4
	performance improvements
	allow KR and KF to be 0
*)
END_FUNCTION_BLOCK

(* POU Mathematical/DIFFER, ST *)
FUNCTION DIFFER : BOOL
VAR_INPUT
	in1 : REAL;
	in2 : REAL;
	X : REAL;
END_VAR


(*
version 1.1	16 mar 2008
programmer 	hugo
tested by		tobias

this function checks if in1 differs more then x from in2
the output is true if abs(in1-in2) > X

*)
DIFFER := ABS(in1 - in2) > X;

(* revision history
hm		8. oct 2006		rev 1.0
	original version

hm		16. mar 2008	rev 1.1
	improverd code for performance

*)
END_FUNCTION

(* POU Time&Date/MULTIME, ST *)
FUNCTION MULTIME : TIME
VAR_INPUT
	t : TIME;
	M : REAL;
END_VAR


(*
version 1.1	14 mar 2008
programmer 	hugo
tested by		tobias

multiplies a time by a real number and returns a time
*)
MULTIME := DWORD_TO_TIME(REAL_TO_DWORD(DWORD_TO_REAL(TIME_TO_DWORD(t))*M));

(* revision history
hm		2. oct 2006	rev 1.0
	original version

hm		14. mar 2008	rev 1.1
	rounded the result after the last digit

*)
END_FUNCTION

(* POU Building/actuators/ACTUATOR_A, ST *)
FUNCTION_BLOCK ACTUATOR_A
VAR_INPUT
	I1 : BYTE;
	IS : BOOL;
	I2 : BYTE;
	RV : BOOL;
	DX : BOOL;
END_VAR
VAR_INPUT CONSTANT
	RUNTIME : TIME;
	SELF_ACT_TIME : TIME;
	OUT_MIN : WORD;
	OUT_MAX : WORD;
END_VAR
VAR_OUTPUT
	Y : WORD;
END_VAR
VAR
	timer : CYCLE_4;
	dx_edge: BOOL;
END_VAR


(*
version 1.0 8. nov. 2008	
programmer 	hugo
tested by	oscat

ACTUATOR_A drives any valve or similar with 0 - 255 continuous control input.
 
*)
(* run the system timer, if self_act_time = t#0s then state is set to 0 *)
timer(T0 := RUNTIME, T1 := RUNTIME, T3 := SELF_ACT_TIME, sl := DX AND NOT dx_edge, sx := 0, S0 := SELF_ACT_TIME > t#0s);
dx_edge := dx;

CASE timer.STATE OF
	0: 	(* self act min value *)
		Y := OUT_MIN;
	1:	(* self_act max value *)
		Y := OUT_MAX;
	3:	(* normal operation *)
		IF rv THEN
			Y := OUT_MAX - (OUT_MAX - OUT_MIN) * SEL(IS, I1, I2) / 255;
		ELSE
			Y := (OUT_MAX - OUT_MIN) * SEL(IS, I1, I2) / 255 + OUT_MIN;
		END_IF;
END_CASE;




(*
hm 	8. nov. 2008	rev 1.0
	original version

*)
END_FUNCTION_BLOCK

(* POU Logic/generators/CYCLE_4, ST *)
FUNCTION_BLOCK CYCLE_4
VAR_INPUT
	E : BOOL := TRUE;
	T0, T1, T2, T3 : TIME;
	S0 : BOOL;
	SX : INT;
	SL : BOOL;
END_VAR
VAR_OUTPUT
	STATE : INT;
END_VAR
VAR
	tx : TIME;
	last : TIME;
	init: BOOL;
END_VAR


(*
version 1.0	
programmer 	hugo
tested by	oscat


 
*)
(* read system timer *)
tx := DWORD_TO_TIME(T_PLC_MS());
(* init on first cycle *)
IF NOT init THEN
	init := TRUE;
	last := tx;
END_IF;

IF E THEN
	IF SL THEN
		(* when sx > 0 then the state sx is forced to start *)
		state:= LIMIT(0,SX,3);
		last := tx;
		(* this is to avoid to reset sx from the calling programm it does work fine on codesys but i am not sure about other systems, because we are writing to an input *)
		SL := FALSE;
	ELSE
		CASE state OF
			0 :	(* wait for T0 and switch to next cycle *)
				IF tx - last >= T0 THEN
					state := 1;
					last := tx;
				END_IF;
			1 : (* wait for T1 over 1st cycle *)
				IF tx - last >= T1 THEN
					state := 2;
					last := tx;
				END_IF;
			2 : (* wait for T1 over 1st cycle *)
				IF tx - last >= T2 THEN
					state := 3;
					last := tx;
				END_IF;
			3 : (* wait for T2 over 2nd cycle *)
				IF tx - last >= T3 THEN
					IF S0 THEN State := 0; END_IF; (* if S0 is false, the sequence stops at state 3 *)
					last := tx;
				END_IF;
		END_CASE;
	END_IF;
ELSE
	state := 0;
	last := tx;
END_IF;



(*
hm	3. nov. 2008	rev 1.0
	original version

*)
END_FUNCTION_BLOCK

(* POU Building/actuators/ACTUATOR_COIL, ST *)
FUNCTION_BLOCK ACTUATOR_COIL
VAR_INPUT
	IN : BOOL;
END_VAR
VAR_INPUT CONSTANT
	self_act_cycle : TIME := t#10d;
	self_act_time : TIME := t#1s;
END_VAR
VAR_OUTPUT
	OUT :BOOL;
	STATUS : BYTE;
END_VAR
VAR
	last : DWORD;
	init: BOOL;
	tx: DWORD;
	now: DWORD;
END_VAR


(*
version 1.0	1. jun. 2008
programmer 	hugo
tested by		tobias

this is an intelligent actuator interface for any coil actuator.
the coil actuator can only switch on/off.
coil actuators like vents can get stuck if they are not u8sed for a long time and need to be autoactivated on ce in a while.

*)
(* read system time *)
now := T_PLC_MS();

(* initialize for first cycle *)
IF NOT init THEN
	last := now;
	init := TRUE;
ELSIF IN THEN
	OUT := TRUE;
	STATUS := 101; (* activated by input *)
	LAST := now;
ELSE
	OUT := FALSE;
	STATUS := 100; (* disabled *)
	(* now we need to check for self activation *)
	tx := now - last;
	IF (self_act_cycle > T#0s) AND (tx >= TIME_TO_DWORD(self_act_cycle)) THEN
		OUT := TRUE;
		STATUS := 102; (* auto activation *)
		IF tx >= TIME_TO_DWORD(self_act_cycle + self_act_time) THEN
			last := now;
			OUT := FALSE;
			STATUS := 100; (* idle *)
		END_IF;
	END_IF;
END_IF;



(*
revision history:

hm		1. jun. 2008 	rev 1.0
	original version

*)
END_FUNCTION_BLOCK

(* POU Building/actuators/ACTUATOR_PUMP, ST *)
FUNCTION_BLOCK ACTUATOR_PUMP
VAR_INPUT
	IN : BOOL;
	MANUAL : BOOL;
	RST : BOOL;
END_VAR
VAR_INPUT CONSTANT
	MIN_ONTIME : TIME := t#10s;
	MIN_OFFTIME : TIME := t#10s;
	RUN_EVERY : TIME := t#10000m;
END_VAR
VAR_OUTPUT
	PUMP : BOOL;
END_VAR
VAR_IN_OUT
	RUNTIME : UDINT;
	CYCLES : UDINT;
END_VAR
VAR
	tx : TIME;
	last_change : TIME;
	meter : ontime;
	old_man : BOOL;
	init: BOOL;
END_VAR

(*
version 1.4		21. oct. 2008
programmer 		oscat
tested BY		oscat

actuator_pump is a pump interface which can be controlled by an input in and an input manual.
in or manual high turns the pump output on.
a rst input is used to reset the runtime counters.
when the pump was not active for a time run_every the actuator turns on the pump automatically for min_ontime.
two setup variables min_ontime and min_offtime guarantee a minimum runtime and offtime of the pump.
the units are hours and the output type is real to prevent from overfow.

*)
tx := DWORD_TO_TIME(T_PLC_MS());

IF NOT init THEN
	init := TRUE;
	last_change := tx;
ELSIF rst THEN
	rst := FALSE;
	runtime := 0;
	cycles := 0;
ELSIF manual AND NOT pump AND NOT old_man THEN
	last_change := tx;
	pump := TRUE;
ELSIF NOT manual AND old_man AND pump AND NOT in THEN
	last_change := tx;
	pump := FALSE;
ELSIF in AND NOT pump AND tx - last_change >= min_offtime THEN
	last_change := tx;
	pump := TRUE;
ELSIF pump AND NOT in AND NOT manual AND tx - last_change >= min_ontime THEN
	last_change := tx;
	pump := FALSE;
ELSIF NOT pump AND (tx - last_change >= run_every) AND (run_every > T#0s) THEN
	last_change := tx;
	pump := TRUE;
END_IF;

meter(in := pump, seconds := runtime, cycles := cycles);
old_man := manual;



(*
hm	27.12.2006		rev 1.1
	fixed a failure while the pump would run for tmin after startup.

hm	15.9.2007		rev 1.2
	replaced Time() with T_PLC_MS for compatibility and performance reasons

hm	13. oct. 2008	rev 1.3
	auto activation can now be disabled when run_every = t#0s

hm	21. oct. 2008	rev 1.4
	changed to use ontime rev 2.0

*)
END_FUNCTION_BLOCK

(* POU Engineering/automation/MANUAL, ST *)
FUNCTION MANUAL : BOOL
VAR_INPUT
	IN : BOOL;
	ON : BOOL;
	OFF : BOOL;
END_VAR


(*
version 1.0	21. nov. 2008
programmer 	hugo
tested by	oscat

MANUAL is a manual override for digital signals.
when on and off = FALSE, the output follows IN.
ON = TRUE forces the output high, and OFF = TRUE forces the output low.


*)
MANUAL := NOT OFF AND (IN OR ON);



(* revision history
hm	21. nov 2008	rev 1.0
	original version


*)
END_FUNCTION

(* POU Engineering/measurements/METER, ST *)
FUNCTION_BLOCK METER
VAR_INPUT
	M1, M2 : REAL;
	I1, I2 : BOOL;
	D : REAL := 1.0;
	RST : BOOL;
END_VAR
VAR_IN_OUT
	MX : REAL;
END_VAR
VAR
	MR : REAL2;
	MX1, MX2 : REAL; (* current consumption value on M1 and M2 *)
	tx: DWORD;
	last: DWORD;
	tc: REAL;
	init: BOOL;
END_VAR

(*
	version 1.4	8. mar. 2009
	programmer 	oscat
	tested BY	oscat

METER measures usage of power or similar values the output MX is the sum of the inputs over time.
MX := sum over time of (I1 * P1 + I2 * P2)/D.
a simple example is the consumption counter for a 2 stage oil burner where stage 1 is 10KW and stage 2 is 20KW.
I1 and I2 decide which value is accounted for, I1 = True only counts P1, I2 is True counts P2 
and I1 and I2 is true counts P1 and P2.
the meter can be used for all kind of consumption meters. P1 and P2 can change on the fly.

*)
(* measure the last cycle time and make sure we onle execute once every millisecond *)
tx := T_PLC_MS();
IF NOT init THEN
	init := TRUE;
	last := tx;
	mr.RX := mx;
	mr.R1 := 0.0;
ELSIF tx = last THEN
	RETURN;
ELSE
	tc := DWORD_TO_REAL(tx - last) * 0.001;
END_IF;
last := tx;

(* reset *)
IF rst THEN
	mr.R1 := 0.0;
	mr.RX := 0.0;
ELSE
	(* current consumption measurement *)
	IF I1 THEN MX1 := M1; ELSE MX1 := 0.0; END_IF;
	IF I2 THEN MX2 := M2; ELSE MX2 := 0.0; END_IF;
	(* add up the current values in a double real *)
	MR := R2_ADD(MR,(SEL(I1,0.0,mx1) + SEL(I2, 0.0, mx2)) / D * TC);
	(* set the current output value *)
	MX := mr.RX;
END_IF;




(* revision history

hm	16. sep.2007		rev 1.0
	original version

hm	7. feb 2008		rev 1.1
	use new version of ft_int to avoid a counting stop at high values
	deleted unnecessary limits

hm	24. mar. 2008	rev 1.2
	use data_type real2 to extend accuracy to 15 digits total
	do not use ft_int which adds unnecessary overhead

hm	8. feb. 2009	rev 1.3
	changed mx to be I/O
	make sure calculation works for cycle times < 1 ms

hm	8. mar. 2009	rev 1.4
	last was not updated
	code improvements

*)
END_FUNCTION_BLOCK

(* POU Mathematical/Double Precision/R2_ADD, ST *)
FUNCTION R2_ADD : REAL2
VAR_INPUT
	X : Real2;
	Y : REAL;
END_VAR
VAR
	temp: REAL;
END_VAR

(*
version 1.0	20. mar. 2008
programmer 	hugo
tested by	tobias

R2_add adds a real to a double real which extends the accuracy of a real to twice as many digits

*)
temp := X.RX;
R2_ADD.RX := Y + X.R1 + X.RX;
R2_ADD.R1 := temp - R2_ADD.RX + Y + X.R1;


(* revision history
hm		20.3.2008	rev 1.0
	original version

*)
END_FUNCTION

(* POU Engineering/measurements/ONTIME, ST *)
FUNCTION_BLOCK ONTIME
VAR_INPUT
	IN : BOOL;
	RST : BOOL;
END_VAR
VAR_IN_OUT
	SECONDS : UDINT;
	CYCLES : UDINT;
END_VAR
VAR
	tx: DWORD;
	last : DWORD;
	edge : BOOL;
	init: BOOL;
	ms: DWORD;
END_VAR

(*
version 2.3	17. dec. 2008
programmer 	oscat
tested by	tobias

ONTIME measures the ontime of a signal in seconds.
the output SECONDS is of type DWORD which results in a total measurement range of 1 second up to 136 years.
internally ontime works with a resolution of milliseconds

*)
(* read system time *)
tx := T_PLC_MS();

(* make sure the first cycle works correctly *)
IF NOT init OR rst THEN
	init := TRUE;
	last := tx;
	SECONDS := 0;
	CYCLES := BOOL_TO_UINT(in);
	ms := 0;
ELSIF IN THEN
	(* add the current milliseconds *)
	ms := (tx - last) + ms;
	IF ms >= 1000 THEN
		seconds := seconds + 1;
		ms := ms - 1000;
	END_IF;
	cycles := cycles + BOOL_TO_UINT(NOT edge);
END_IF;
last := tx;
edge := in;


(* revision history
hm 22.2.2007		rev 1.1
	changed VAR RETAIN PERSISTENT to VAR RETAIN for better compatibility
	wago lon contollers do not support persisitent

hm 2.8.2007		rev 1.2
	adding time up in a real number will automatically lead to the point where 
	small time scales like the cycle time will be below the resolution of real and therefore
	ontime would not increase in small steps as necessary
	the time is now measured internally in two  dwords and be converted to real only for
	output purposes.
	deleted the variable power because it was unnecessary

hm	16.9.2007		rev 1.3
	changes time() to T_plc_ms() for compatibility reasons

hm	2. dec. 2007	rev 1.4
	chaged code for better performance

hm	16. mar. 2008	rev 1.5
	added type conversions to avoid warnings under codesys 3.0

hm	21. oct. 2008	rev 2.0
	changed module for much better performance and allow for external result storage

hm	10. nov. 2008	rev 2.1
	increased internal resolution to milliseconds

hm	16. nov. 2008	rev 2.2
	changed typecast to avoid warnings

hm	17. dec. 2008	rev 2.3
	fixed an error when in would be true for more then 49 days
*)
END_FUNCTION_BLOCK

(* POU Building/actuators/ACTUATOR_UD, ST *)
FUNCTION_BLOCK ACTUATOR_UD
VAR_INPUT
	UD : BOOL;
	ON : BOOL;
	Manual : BOOL;
	Up : BOOL;
	Dn : BOOL;
	off : BOOL;
	YUP_in : BOOL;
	YDN_in : BOOL;
END_VAR
VAR_INPUT CONSTANT
	TON : TIME;
	TOFF : TIME;
	out_return : BOOL;
END_VAR
VAR_OUTPUT
	Yup : BOOL;
	Ydn : BOOL;
	status : BYTE;
END_VAR
VAR
	tx : TIME;
	last : TIME;
	init: BOOL;
END_VAR

(*
version 1.3	17. oct. 2008
programmer 	hugo
tested by		tobias

out_ud is a up/dn or Right/left locked output driver.
it can be controlled by automatic inputs UD and ON as well as manual inputs for up and dn.
a security input to shut off at any time is prvided by the off input.
two time set inputs ton and toff specify a minimum on time for outputs and a minimum off time before the next output can become active.
the module assures that only one output can be active at any time.
for higher security pls make sure you use hardware locking of the outputs to prevent from defective wiring or outputs.
further security is provided b feedback inputs Yup_in and Ydn_in which are separate inputs for the output signal, if these inputs are not available 
pls connect them directly to Yup and Ydn.
manual mode will override automatic mode by setting the manual input high.
a status output will be 0 for normal operation or 1 - 99 for error reporting and 101 - 199 for status reporting
The status output is ESR comptible.
*)
(* read system time *)
tx := DWORD_TO_TIME(T_PLC_MS());

IF NOT init THEN
	(* INITIALIZATION AT FIRST CALL *)
	last := tx;
	init := TRUE;
ELSIF off THEN
	(* emergency shut off detected *)
	Yup := FALSE;
	ydn := FALSE;
	last := tx;
	status := 101;

(* Watch FOR MIN TON TIME *)
ELSIF ((Yup OR Ydn) AND tx - last < Ton) THEN
	RETURN;
ELSIF NOT yup AND NOT ydn AND tx - last < toff THEN
	RETURN;

(* manual operation *)
ELSIF manual THEN
	status := 102;
	(* directional chage set both outs 0 first *)
	IF yup AND NOT up OR ydn AND NOT dn THEN
		ydn := FALSE;
		yup := FALSE;
		last := tx;
	(* manual up operation *)
	ELSIF UP AND NOT DN AND NOT OFF THEN
		Ydn := FALSE;
		Yup := TRUE;
		last := tx;
		status := 103;
	(* manual down operation *)
	ELSIF DN AND NOT UP AND NOT OFF THEN
		Yup := FALSE;
		Ydn := TRUE;
		last := tx;
		status := 104;
	(* maual mode but no up or down *)
	ELSE
		IF YUP OR YDN THEN LAST := tx; END_IF;
		Yup := FALSE;
		ydn := FALSE;
	END_IF;

(* automatic operation *)
ELSE
	(* directional change set outputs low first *)
	IF yup AND NOT ud OR ydn AND UD THEN
		yup := FALSE;
		ydn := FALSE;
		last := tx;
	(* automatic up operation *)
	ELSIF Ud AND on AND NOT OFF THEN
		Ydn := FALSE;
		Yup := TRUE;
		last := tx;
		status := 111;

	(* automatic down operation *)
	ELSIF NOT UD AND on AND NOT OFF THEN
		Yup := FALSE;
		Ydn := TRUE;
		last := tx;
		status := 112;
	(* standby mode *)
	ELSE
		IF Yup OR Ydn THEN last := tx; END_IF;
		Yup := FALSE;
		Ydn := FALSE;
		status := 110;
	END_IF;
END_IF;

(* make sure Yup and Ydn are never on at the same time *)
IF Ydn AND Yup_in AND out_return THEN
	Ydn := FALSE;
	status := 1;
END_IF;
IF Yup AND Ydn_in AND out_return THEN
	Yup := FALSE;
	status := 2;
END_IF;



(* revision history
hm 22. jan 2007	rev 1.1
	added status output
	changed inputs ton, toff to config variables
	added config var out_return to enable yup_in and Ydn_in
	manual mod will override automatic mode 

hm	15.9.2007	rev 1.2
	replaced Time() with T_PLC_MS for compatibility and performance reasons

hm	17. oct. 2008	rev 1.3
	deleted unnecessary initialization with 0
*)
END_FUNCTION_BLOCK

(* POU Building/electrical/CLICK, ST *)
FUNCTION_BLOCK CLICK
VAR_INPUT
	in : BOOL;
END_VAR
VAR_OUTPUT
	Q : BOOL;
	single : BOOL;
	double : BOOL;
	triple : BOOL;
	status: BYTE;
END_VAR
VAR_INPUT CONSTANT
	T_debounce : TIME := t#10ms;
	T_short : TIME := t#200ms;
	T_pause : TIME := t#500ms;
	T_reconfig : TIME := t#1m;
END_VAR
VAR
	s_in : SW_RECONFIG;
	tx: TIME;
	state: INT;
	last: TIME;
END_VAR

(*
version 2.0	28. dec. 2008
programmer 	oscat
tested by		oscat

click checks an input for single, double or tripple click and sets the corresponding output single, doulbe or triple for the time the input stays high at the last click.
the maximum high and low time for a click can be configured with setup variables.
the input configures itself to be high or low active depending on which state the input stays longer than t_reconfig.

*)
(* reconfiguration and debounce circuitry *)
s_in(in := in, TD := T_debounce, TR := T_reconfig);

(* read system time *)
tx := DWORD_TO_TIME(T_PLC_MS());

(* count the mumber of clicks *)
IF s_in.Q XOR Q THEN
	last := tx;
	IF s_in.Q THEN state := state + 1; END_IF;
END_IF;
Q := s_in.Q;

(* set outputs *)
IF state > 0 THEN
	IF (Q AND tx - last > t_short) OR (NOT Q AND tx - last > t_pause) THEN
		CASE state OF
			1:	single := TRUE;
				status := 111;
			2:	double := TRUE;
				status := 112;
			3:	triple := TRUE;
				status := 113;
		END_CASE;
		state := 0;
	END_IF;
ELSIF NOT q THEN
	single := FALSE;
	double := FALSE;
	triple := FALSE;
	status := 110;
	last := tx;
	state := 0;
END_IF;





(* revision history

15 Feb 2007	rev 1.0	hm
	created original version

18.5.2007	rev 1.1 hm
	corrected an error while execution would stop after t_reconfig elapsed.

15.9.2007	rev 1.2 hm
	replaced Time() with T_PLC_MS for compatibility and performance reasons

28. dec. 2008	rev 2.0
	rewritten using modular approach

*)
END_FUNCTION_BLOCK

(* POU Building/electrical/SW_RECONFIG, ST *)
FUNCTION_BLOCK SW_RECONFIG
VAR_INPUT
	IN : BOOL;
	TD : TIME;
	TR : TIME;
END_VAR
VAR_OUTPUT
	Q : BOOL;
END_VAR
VAR
	T1, T2 : TON;
	INV: BOOL;
END_VAR


(*
version 1.0	22. oct. 2008
programmer 	hugo
tested by	oscat

SW_reconfig detects if an input is high or low active and debounces the input

*)
(* run debounce circuit *)
t1(in := IN, PT := TD);

IF tr > t#0s THEN
	(* generate output *)
	Q := t1.Q XOR inv;
	(* reconfiguration timer *)
	T2(in := Q, pt := TR);
	(* when T2.Q goes high then reverse INV *)
	IF T2.Q THEN INV := NOT INV; END_IF;
ELSE
	Q := t1.Q;
END_IF;



(* revision history
hm	22.10.2008	rev 1.0
	original version

*)
END_FUNCTION_BLOCK

(* POU Mathematical/INV, ST *)
FUNCTION INV : REAL
VAR_INPUT
	X : REAL;
END_VAR


(*
version 1.1	10. mar. 2009
programmer 	hugo
tested by		tobias

This function calculates the result of 1 / X

*)
IF X <> 0.0 THEN INV := 1.0 / X; END_IF;




(* revision history
hm	26. oct. 2008	rev 1.0
	original version

hm	10. mar. 2009	rev 1.1
	real constants updated to new systax using dot

*)
END_FUNCTION

(* POU Building/electrical/CLICK_MODE, ST *)
FUNCTION_BLOCK CLICK_MODE
VAR_INPUT
	IN : BOOL;
END_VAR
VAR_OUTPUT
	SINGLE : BOOL;
	DOUBLE : BOOL;
	LONG : BOOL;
	TP_LONG : BOOL;
END_VAR
VAR_INPUT CONSTANT
	T_LONG : TIME := t#500ms;
END_VAR
VAR
	Timer : TP;
	cnt : INT;
	last : BOOL;
END_VAR


(*
version 1.0	13. nov. 2008
programmer 	oscat
tested by	hugo

click_mode decodes an input for single, double or long click and sets the corresponding output single, doulbe or long.
the input configures itself to be high or low active depending on which state the input stays longer than t_reconfig.

*)
(* when input goes high start the timer to decode pulses *)
timer(in := IN, PT := T_LONG);
single := FALSE;
double := FALSE;

IF timer.Q THEN
	(* decode pulses while the timer is active *)
	IF NOT in AND last THEN	cnt := cnt + 1; END_IF;
ELSE
	CASE cnt OF
		1 : single := TRUE;
		2 : double := TRUE;
	END_CASE;
	cnt := 0;
END_IF;
last := in;
TP_LONG := NOT timer.Q AND (NOT LONG) AND IN;
LONG := NOT timer.Q AND in;




(* revision history

hm	13. nov. 2008	rev 1.0
	original release

*)
END_FUNCTION_BLOCK

(* POU Building/electrical/DEBOUNCE, ST *)
FUNCTION_BLOCK DEBOUNCE
VAR_INPUT
	IN : BOOL;
	TD : TIME;
	PM : BOOL;
END_VAR

VAR_OUTPUT
	Q : BOOL;
END_VAR
VAR
	deb : TOF;
END_VAR

(*
version 1.0	22. sep. 2008
programmer 	oscat
tested by	tobias

DEBOUNCE is used to debounce switch inputs.
in addition to the debounce functionality this FB can also be used to detect rising edges on IN when PM = TRUE.
When PM = FALSE, Q follows in with the debounce functionality.

*)
IF NOT deb.Q AND IN THEN
	(* rising edge on input detetced a *)
	Q := TRUE;
ELSIF NOT PM THEN
	Q := deb.Q;
ELSE
	Q := FALSE;
END_IF;

(* run debounce timer *)
deb(IN := IN, PT := TD);



(*
hm 22. sep. 2008	rev 1.0
	original version

*)
END_FUNCTION_BLOCK

(* POU Building/electrical/DIMM_2, ST *)
FUNCTION_BLOCK DIMM_2
VAR_INPUT
	SET : BOOL;
	VAL : BYTE := 255;
	I1 : BOOL;
	I2 : BOOL;
	RST : BOOL;
END_VAR
VAR_INPUT CONSTANT
	T_DEBOUNCE : TIME := T#10ms;
	T_ON_MAX : TIME := T#0h;
	T_DIMM_START : TIME := T#1s;
	T_DIMM: TIME := T#3s;
	MIN_ON : BYTE := 50;
	MAX_ON : BYTE := 255;
	RST_OUT : BOOL := TRUE;
	SOFT_DIMM : BOOL := TRUE;
	DBL1_TOG : BOOL;
	DBL2_TOG : BOOL;
	DBL1_SET : BOOL;
	DBL2_SET : BOOL;
	DBL1_POS : BYTE;
	DBL2_POS : BYTE;
END_VAR
VAR_OUTPUT
	Q : BOOL := FALSE;
	D1 : BOOL;
	D2 : BOOL;
END_VAR
VAR_IN_OUT
	OUT : BYTE;
END_VAR
VAR
	t1, t2 : TOF;
	dc1, dc2 : CLICK_MODE;
	t3 : TON;
	dim : _RMP_B;
END_VAR

(*
version 1.0	22. mar. 2009
programmer 	hugo
tested by	tobias

this is an intelligent dimmer interface with an autoset feature using double switch inputs
a configurable debounce timer will debounce the input signals
if t_on_max is set to anything other then 0 the output will be turned off after the max on time is reached.
the times for debounce, dimming ramp, wait time before dimming and max on time are all programmable.

the dimmer has outputs Q for on and off and also out with the analog dimm value.
two additional outputs d1 and d2 decode double clicks on i1 and i2.

*)
(* debouncing for inputs i1 and i2 *)
t1(IN := I1, PT := T_DEBOUNCE);
t2(IN := I2, PT := T_DEBOUNCE);
dc1(in := t1.Q, T_LONG := T_DIMM_START);
dc2(in := t2.Q, T_LONG := T_DIMM_START);


IF RST THEN
	IF RST_OUT THEN out := 0; END_IF;
	Q := FALSE;
	D1 := FALSE;
	D2 := FALSE;
ELSIF set THEN
	OUT := VAL;
	Q := TRUE;
ELSIF dc1.SINGLE THEN
	(* single click on i1 turns the dimmer on *)
	out := LIMIT(MAX(MIN_ON,1), out, MAX_ON);
	Q := TRUE;
ELSIF dc2.SINGLE THEN
	(* single click on i2 turns the dimmer off *)
	Q := FALSE;
ELSIF dc1.TP_LONG THEN
	(* continuous on at i1 dimms up *)
	IF NOT Q THEN
		out := SEL(SOFT_DIMM, LIMIT(MAX(MIN_ON,1), out, MAX_ON), 1);
	END_IF;
	Q := TRUE;
	dim.DIR := TRUE;
ELSIF dc2.TP_LONG THEN
	(* continuous on at i2 dimms down *)
	dim.DIR := FALSE;
END_IF;

(* set the double click output *)
IF NOT DBL1_TOG THEN D1 := FALSE; END_IF;
IF dc1.DOUBLE THEN
	IF DBL1_SET THEN
		OUT := DBL1_POS;
		Q := TRUE;
	ELSE
		D1 := NOT D1;
	END_IF;
END_IF;
IF NOT DBL2_TOG THEN D2 := FALSE; END_IF;
IF dc2.DOUBLE THEN
	IF DBL2_SET THEN
		OUT := DBL2_POS;
		Q := TRUE;
	ELSE
		D2 := NOT D2;
	END_IF;
END_IF;


(* while dimming is active ramp the output out up or down *)
dim(dir := dc2.LONG, e := dc1.LONG OR dc2.LONG , TR := T_DIMM, rmp := out);

(* turn off output if a value of 0 is reached *)
IF out = 0 THEN Q := FALSE; END_IF;

(* limit the maximum runtime *)
IF t_ON_MAX > t#0s THEN
	t3(in := q, pt := T_ON_MAX);
	Q := Q XOR t3.Q;
END_IF;




(* revision history

hm 22. mar. 2009	rev 1.0
	original version

*)
END_FUNCTION_BLOCK

(* POU Building/electrical/DIMM_I, ST *)
FUNCTION_BLOCK DIMM_I
VAR_INPUT
	SET : BOOL;
	VAL : BYTE := 255;
	IN : BOOL;
	RST : BOOL;
END_VAR
VAR_INPUT CONSTANT
	T_DEBOUNCE : TIME := T#10ms;
	T_RECONFIG : TIME := T#10s;
	T_ON_MAX : TIME := T#0h;
	T_DIMM_START : TIME := T#1s;
	T_DIMM: TIME := T#3s;
	MIN_ON : BYTE := 50;
	MAX_ON : BYTE := 255;
	SOFT_DIMM : BOOL := TRUE;
	DBL_toggle : BOOL;
	RST_OUT : BOOL;
END_VAR
VAR_OUTPUT
	Q : BOOL := FALSE;
	DBL : BOOL;
END_VAR
VAR_IN_OUT
	OUT : BYTE;
END_VAR
VAR
	config : SW_RECONFIG;
	decode : CLICK_MODE;
	t3 : TON;
	dim : _RMP_B;
	dir : BOOL;
END_VAR

(*
version 2.3	26. jan. 2009
programmer 	hugo
tested by		tobias

this is an intelligent dimmer interface with an autoset feature for "in" it will automatically detect the type of switch:
low active pulses or high high active pulses are allowd for in.
a configurable debounce timer will debounce input signals
if t_on_max is set to anything other then 0 the output will be turned off after the max on time is reached.
the times for debounce, dimming ramp, wait time before dimming and max on time are all programmable.

the dimmer has outputs Q for on and off and also out with the analog dimm value.

*)
(* the input is first sent through auto reconfiguration and debouncing *)
config(IN := IN, TD := T_DEBOUNCE, TR := T_RECONFIG);
decode(in := config.Q, T_LONG := T_DIMM_START);

IF RST THEN
	IF rst_out THEN out := 0; END_IF;
	Q := FALSE;
	dir := out > 127;
ELSIF set THEN
	out := val;
	Q := TRUE;
	(* set direction to up when value < 127 otherwise set dir down dir is reversed because next action will reverse again *)
	dir := out > 127;
ELSIF decode.SINGLE THEN
	(* a single click reverses output Q *)
	Q := NOT Q;
	(* when dimmer is turned on we need to limit out to min and max limits *)
	IF Q THEN	out := LIMIT(MAX(MIN_ON,1), out, MAX_ON);	END_IF;
	(* set the appropriate direction of dimmer dir is reversed because next action will reverse again *)
	dir := out > 127;
ELSIF decode.TP_LONG THEN
	IF NOT Q THEN
		IF SOFT_DIMM THEN
			OUT := 1;
			dir := TRUE;
		ELSE
			OUT := LIMIT(MAX(MIN_ON,1), out, MAX_ON);
			DIR := out < 127;
		END_IF;
		Q := TRUE;
	ELSE
		(* reverse direction with every long click *)
		dir := NOT dir;
	END_IF;
END_IF;

(* set the double click output *)
IF NOT dbl_toggle THEN dbl := FALSE; END_IF;
IF decode.DOUBLE THEN dbl := NOT dbl; END_IF;

(* while dimming is active ramp the output out up or down *)
dim(DIR := dir, e := decode.LONG AND Q, TR := T_DIMM, rmp := out);

(* reverse direction when limits are reached *)
IF out = 0 THEN
	dir := TRUE;
ELSIF out = 255 THEN
	dir := FALSE;
END_IF;

(* limit the maximum runtime *)
IF t_ON_MAX > t#0s THEN
	t3(in := q, pt := T_ON_MAX);
	Q := Q XOR t3.Q;
END_IF;




(* revision history

hm 22.1.2007		rev 1.1
	deleted unused structure ramp

hm 2.feb 2007		rev 1.2
	changed structure to read time() at the beginning for better time consistency if a higher priorized tak interrupts dimm_i
	added statements in case structure for state 1 to allow for short 1 cycle input pulses

hm 	15.9.2007		rev 1.3
	replaced Time() with T_PLC_MS for compatibility and performance reasons

hm	30. sep. 2008	rev 1.4
	added Input VAL to supply value for set input
	added setup parameter init_val

hm	22. oct. 2008	rev 2.0
	new code and features

hm	14. nov. 2008	rev 2.1
	added soft_dimm feature

hm	16. nov. 2008	rev 2.2
	added reset out feature

hm	26. jan. 2009	rev 2.3
	dimming will also reverse at out = 0
	rst will override set
*)
END_FUNCTION_BLOCK

(* POU Building/electrical/F_LAMP, ST *)
FUNCTION_BLOCK F_LAMP
VAR_INPUT
	SWITCH : BOOL;
	DIMM : BYTE := 255;
	RST : BOOL;
END_VAR
VAR_OUTPUT
	LAMP : BYTE;
	STATUS : BYTE;
END_VAR
VAR_IN_OUT
	ONTIME : UDINT;
	CYCLES : UDINT;
END_VAR
VAR_INPUT CONSTANT
	T_NO_DIMM : UINT := 100;
	T_MAINTENANCE : UINT := 15000;
END_VAR
VAR
	runtime : ONTIME;
END_VAR

(*
version 1.2	22. oct. 2008
programmer 	hugo
tested by	oscat

F_Lamp is an interface to flourescent lamps. its main purpose is to protect flourescent lamps from dimming within the first T_NO_DIMM Time.
If Flourescent Lamps are dimmed during the first 100 hours the lifetime of the lamp is reduced dramatically.
The interface also counts ontime and cycles of the lamp for maintanance purposes.

*)
runtime(in := switch, seconds := ontime, cycles := cycles);

IF RST THEN
	ONTIME := 0;
	CYCLES := 0;
END_IF;
IF SWITCH THEN
	IF ontime < T_NO_DIMM * 3600 THEN
		LAMP := 255;
		STATUS := 111;
	ELSE
		LAMP := DIMM;
		STATUS := 112;
	END_IF;
ELSE
	LAMP := 0;
	STATUS := 110;
END_IF;


IF ontime >= T_maintenance * 3600 AND T_Maintenance > 0 THEN
	status := 120;
END_IF;



(* revision history
hm	8. feb. 2007	rev 1.1
	original version

hm	22. oct. 2008	rev 1.2
	changed use of ontime for ontime 2.0
	ontime is now in seconds not hours
*)
END_FUNCTION_BLOCK

(* POU Building/electrical/PULSE_LENGTH, ST *)
FUNCTION_BLOCK PULSE_LENGTH
VAR_INPUT
	in : BOOL;
END_VAR
VAR_OUTPUT
	short : BOOL;
	middle : BOOL;
	long : BOOL;
END_VAR
VAR_INPUT CONSTANT
	T_short : TIME := t#100ms;
	T_long : TIME := t#1s;
END_VAR
VAR
	tx : TIME;
	tn: TIME;
	edge : BOOL;
END_VAR

(*
version 1.1	15 sep 2007
programmer 	oscat
tested by	oscat

Pulse_length indicates on 3 outputs if an input pulse had been shorter than T_short (short = True), longer than T_long (long = True) or between T_short and T_long (middle = True).

*)
(* read system time *)
tx := DWORD_TO_TIME(T_PLC_MS());

(* reset outputs, they should only be active 1 cycle *)
short := FALSE;
Middle := FALSE;
long := FALSE;

(* detect rising edge *)
IF in AND NOT edge THEN
	edge := TRUE;
	tn := tx;

(* detect for falling edge *)
ELSIF NOT in AND edge THEN
	edge := FALSE;
	tn := tx - tn;
	IF tn < t_short THEN
		short := TRUE;
	ELSIF tn > t_long THEN
		long := TRUE;
	ELSE
		Middle := TRUE;
	END_IF;

(* generate long pulse as soon as T_long is reached *)
ELSIF in AND tx - tn > t_long THEN
	long := TRUE;
END_IF;


(* revision history

hm	15. feb 2006	rev 1.0
	original version

hm	15 sep 2007		rev 1.1
	replaced Time() with T_PLC_MS for compatibility and performance reasons

*)
END_FUNCTION_BLOCK

(* POU Building/electrical/PULSE_T, ST *)
FUNCTION_BLOCK PULSE_T
VAR_INPUT
	IN : BOOL;
	T1 : TIME;
	T2 : TIME;
	RST : BOOL;
END_VAR
VAR_OUTPUT
	Q : BOOL;
END_VAR
VAR
	init: BOOL;
	last: TIME;
	tx: TIME;
	edge: BOOL;
END_VAR


(*
version 1.0	15. jul. 2008
programmer 	hugo
tested by	oscat

PULSE_T generates a pulse of length T2 if the input pulse is shorter than T1.
if the input pulse is longer than T1, the output follows the input.
and rising edge on in will kill a possible output pulse and generate a new pulse instead.

*)
tx := DWORD_TO_TIME(T_PLC_MS());
IF NOT init THEN
	init := TRUE;
	last := tx;
ELSIF RST THEN
	(* asynchronous reset *)
	Q := FALSE;
ELSIF IN AND NOT edge AND NOT Q THEN
	(* a rising edge on in will reversre the output status, if new pulse is startet the start time is stored in last *)
	last := tx;
	Q := TRUE;
ELSIF NOT IN AND edge AND ((tx - last) > T1) THEN
	(* a falling edge on IN will clear the output if in was high for more then T1 *)
	Q := FALSE;
ELSIF (tx - last) >= T2 THEN
	(* timeout for long pulse if second click did not occur or in stays high *)
	Q := FALSE;
END_IF;

edge := IN;

(* revision histroy
hm	15. jul. 2008	rev 1.0
	original release


*)	
END_FUNCTION_BLOCK

(* POU Building/electrical/SWITCH_I, ST *)
FUNCTION_BLOCK SWITCH_I
VAR_INPUT
	set : BOOL;
	in : BOOL;
	rst : BOOL;
END_VAR
VAR_INPUT CONSTANT
	T_debounce : TIME := T#10ms;
	T_reconfig : TIME := T#1s;
	T_on_max : TIME := T#0h;
END_VAR
VAR_OUTPUT
	Q : BOOL;
END_VAR
VAR
	state : BYTE;
	edge : BOOL;
	r_edge : BOOL;
	T_on : TIME;
	tx: TIME;
END_VAR

(*
version 1.1	15 sep 2007
programmer 	oscat
tested by	oscat

this is an intelligent switch interface which has an autodetect feature for in and it will detect the type of switch connected automatically
the input can be connected to low active pulses, high active pulses and on/off switch.
it will automatically adjust to the correct type without manual adjustment
a configurable debounce timer will debounce input signals
if t_on_max is set to anything other then 0 the output will be turned off after the max on time is reached.

*)
(* read system time *)
tx := DWORD_TO_TIME(T_PLC_MS());

(* asynchronous set and reset first *)
IF set AND NOT rst THEN
	Q := TRUE;
	T_on := tx;
ELSIF rst THEN
	Q := FALSE;
(* check FOR input edge AND start debounce timer *)
ELSIF (in XOR edge) AND NOT (state = 1) THEN
	state := 1;
	T_on := Tx;
(* edge was detected and debounce time elapsed *)
ELSIF (state = 1) AND (Tx - t_debounce >= T_on) THEN
	state := 2;
	(* react on rising or falling edge depending on r_edge *)
	IF r_edge XOR in THEN Q := NOT Q; END_IF;
(* wait for T_reconfig and adjust r_edge *)
ELSIF state = 2 AND Tx - t_reconfig >= T_on THEN
	r_edge := in;
END_IF;
IF Q AND T_on_max > t#0ms AND Tx >= T_on + T_on_max THEN
	Q := FALSE;
END_IF;
edge := in;

(* revision history

hm	4 aug 2006	rev 1.0
	original version

hm	15.9.2007	rev 1.1
	replaced Time() with T_PLC_MS for compatibility and performance reasons

*)
END_FUNCTION_BLOCK

(* POU Building/electrical/SWITCH_X, ST *)
FUNCTION_BLOCK SWITCH_X
VAR_INPUT
	IN1 : BOOL;
	IN2 : BOOL;
	IN3 : BOOL;
	IN4 : BOOL;
	IN5 : BOOL;
	IN6 : BOOL;
END_VAR
VAR_OUTPUT
	Q1 : BOOL;
	Q2 : BOOL;
	Q3 : BOOL;
	Q4 : BOOL;
	Q5 : BOOL;
	Q6 : BOOL;
	Q31 : BOOL;
	Q41 : BOOL;
	Q51 : BOOL;
	Q61 : BOOL;
	Q32 : BOOL;
	Q42 : BOOL;
	Q52 : BOOL;
	Q62 : BOOL;
END_VAR
VAR_INPUT CONSTANT
	t_debounce : TIME := t#50ms;
END_VAR
VAR
	init : BOOL;
	T1, T2, T3, T4, T5, T6 : TOF;
	tx: TIME;
	x1: BOOL;
	x2: BOOL;
	E1, E2 : BOOL;
END_VAR

(*
version 1.0	15 Feb 2007
programmer 	oscat
tested by	oscat

*)
(* initialize on startup *)
IF NOT init THEN
	init := TRUE;
	IF t_debounce < t#50ms THEN tx := t#50ms; ELSE tx := t_debounce; END_IF;
	T1(PT := Tx);
	T2(PT := Tx);
	T3(PT := Tx);
	T4(PT := Tx);
	T5(PT := Tx);
	T6(PT := Tx);
ELSE
	Q1 := FALSE;
	Q2 := FALSE;
	Q3 := FALSE;
	Q4 := FALSE;
	Q5 := FALSE;
	Q6 := FALSE;
	Q31 := FALSE;
	Q41 := FALSE;
	Q51 := FALSE;
	Q61 := FALSE;
	Q32 := FALSE;
	Q42 := FALSE;
	Q52 := FALSE;
	Q62 := FALSE;
END_IF;

(* read inputs and debounce *)
	T1(IN := IN1);
	T2(IN := IN2);
	T3(IN := IN3);
	T4(IN := IN4);
	T5(IN := IN5);
	T6(IN := IN6);

(* detect edge of IN1 and IN2 *)
IF t1.Q AND NOT E1 THEN X1 := TRUE; END_IF;
IF t2.Q AND NOT E2 THEN X2 := TRUE; END_IF;

IF t1.Q THEN
	IF t3.q THEN
		q31 := TRUE;
		X1 := FALSE;
	ELSIF t4.q THEN
		q41 := TRUE;
		X1 := FALSE;
	ELSIF t5.q THEN
		q51 := TRUE;
		X1 := FALSE;
	ELSIF t6.q THEN
		q61 := TRUE;
		X1 := FALSE;
	END_IF;
ELSIF t2.Q THEN
	IF t3.q THEN
		q32 := TRUE;
		X2 := FALSE;
	ELSIF t4.q THEN
		q42 := TRUE;
		X2 := FALSE;
	ELSIF t5.q THEN
		q52 := TRUE;
		X2 := FALSE;
	ELSIF t6.q THEN
		q62 := TRUE;
		X2 := FALSE;
	END_IF;
(* in1 was active alone *)
ELSIF NOT T1.Q AND E1 AND X1 THEN
	Q1 := TRUE;
	X1 := FALSE;
ELSIF NOT T2.Q AND E2 AND X2 THEN
	Q2 := TRUE;
	X2 := FALSE;
ELSIF T3.Q THEN
	Q3 := TRUE;
ELSIF T4.Q THEN
	Q4 := TRUE;
ELSIF T5.Q THEN
	Q5 := TRUE;
ELSIF T6.Q THEN
	Q6 := TRUE;
END_IF;

(* save state of in1 and in2 *)
E1 := T1.Q;
E2 := T2.Q;
END_FUNCTION_BLOCK

(* POU Building/electrical/TIMER_1, ST *)
FUNCTION_BLOCK TIMER_1
VAR_INPUT
	E : BOOL := TRUE;
	DTI : DT;
	START : TOD;
	DURATION : TIME;
	DAY : BYTE := 2#0111_1111;
END_VAR
VAR_OUTPUT
	Q : BOOL;
END_VAR
VAR
	td : DATE;
	tdt : DT;
END_VAR

(*
version 2.1	6. nov. 2008
programmer 	oscat
tested by	oscat

this is a simple timer that generates an output pulse on selected days.
the output pulse width can be programmed with duration, if set to 0 no pulse is generated.
day specifies the specific days for the event to occur, bit 0 = sunday, bit 1 = saturday, bit 2 = friday ....
for all days to be active 127 has to be specified for DAY.

*)
td := DT_TO_DATE(DTI);
tdt := DATE_TO_DT(td) + TOD_TO_TIME(start);

Q := DTI >= tdt AND dti < tdt + duration AND E AND (SHR(BYTE#128, DAY_OF_WEEK(td)) AND day) > 0;



(*
1.12.2006 hm		rev 1.1
	corrected an error with pulse width = 0.

25.12.2006 hm		rev 1.2
	corrected an error when timer overflows.

14.apr 2007 hm		rev 1.3
	corrected an error while while output would not go active when start year would be 1970.
	increase accuracy by checking every 100ms
	added init section to compensate for timer overflow

15.9.2007 hm		rev 1.4
	replaced Time() with T_PLC_MS for compatibility and performance reasons

hm	1. okt 2007		rev 1.5
	corrected an error while output would not stay active over midnight.

hm	17. jan 2008	rev 1.6
	New code with better performance  
	Output is now only active during the time of day it is supposed to 
	no pulse is generated at power up

hm	7. oct. 2008	rev 1.7
	changed function weekday to day_of_week

hm	23. oct. 2008	rev 2.0
	new code, added input E, now days can be selected by bits in byte day

hm	6. nov. 2008	rev 2.1
	added default for input EN and input DAY
*)
END_FUNCTION_BLOCK

(* POU Time&Date/DAY_OF_WEEK, ST *)
FUNCTION DAY_OF_WEEK : INT
VAR_INPUT
	IDATE : DATE;
END_VAR


(*
version 1.4	7. oct. 2008
programmer 	hugo
tested by	tobias

calculates the weekday of a week according to ISO8601   
monday = 1 ..... sunday = 7  

*)
DAY_OF_WEEK := DWORD_TO_INT((DATE_TO_DWORD(idate) / 86400+3) MOD 7) + 1;



(* revision history
hm 	21.8.06 		rev 1.1
	corrected a miscalculation

hm	23.12.2007		rev 1.2
	correction for step7

hm	7. apr. 2008	rev 1.3
	deleted unused step7 code

hm	7. oct. 2008	rev 1.4
	changed name of function from weekday to day_of_week

*)
END_FUNCTION

(* POU Building/electrical/TIMER_2, ST *)
FUNCTION_BLOCK TIMER_2
VAR_INPUT
	DT_in : DT;
	start : TOD;
	duration : TIME;
	mode : BYTE;
	HOLIDAY : BOOL;
END_VAR
VAR_OUTPUT
	Q : BOOL;
END_VAR
VAR
	last_check : TIME;
	dat : DATE;
	daytime : TOD;
	activation: TIME;
	tx: TIME;
	enabled: BOOL;
	init: BOOL;
	wday : INT;
END_VAR

VAR RETAIN
	run_date : DATE;
END_VAR

(*
version 1.4	20. oct. 2008
programmer 	oscat
tested by	oscat

this timer generated programmabe output pulses per day, week, month and so on.
the mode input determines on which days the timer will be active.
	mode = 0			never
	mode = 1..7			monday .. sunday
	mode = 11			every day
	mode = 12			every second day
	mode = 13			every 3rd day
	mode = 14			every 4th day
	mode = 15			every 5th day
	mode = 16 			every 6th day
	mode = 20			only monday - friday
	mode = 21			only sat - sunday
	mode = 22			workdays only
	mode = 23			holidays and weekend
	mode = 24			holidays only
	mode = 25			every 1st day of the month
	mode = 26			every last day of the month
	mode = 27			every 31 of december
	mode = 28			every 1st of january

a holiday input can be used to supply holiday information to the module.
*)
(* read system time *)
tx := DWORD_TO_TIME(T_PLC_MS());

IF NOT init THEN
	init := TRUE;
	last_check := tx - t#100ms;
END_IF;

(* for performance resons exit if execution is not necessary *)
IF tx - last_check < T#100ms THEN RETURN; END_IF;

(* calculate temp variables *)
dat := DT_TO_DATE(dt_in);
daytime := DT_TO_TOD(dt_in);
wday := DAY_OF_WEEK(dat);

(* calculate if any action is necessary today *)
CASE mode OF
	1..7:	(* mondays to fridays *)
		enabled := wday = BYTE_TO_INT(mode);
	11:	(* every day *)
		enabled := TRUE;
	12..16:	(* every nth day *)
		enabled := (DATE_TO_DWORD(dat)/86400) MOD (mode - 10) = 0;
	20:	(* monday - friday *)
		enabled := wday <= 5;
	21:	(* saturday and sunday *)
		enabled := wday > 5;
	22: (* workdays only *)
		enabled := wday <= 5 AND NOT holiday;
	23:	(* holidays and weekends *)
		enabled := wday > 5 OR holiday;
	24:	(* holidays only *)
		enabled := holiday;
	25:	(* 1st day of the month *)
		enabled := DAY_OF_MONTH(dat) = 1;
	26:	(* last day of month *)
		enabled := DAY_OF_MONTH(dat + t#1d) = 1;
	27:	(* 31st of december *)
		enabled := DAY_OF_MONTH(dat) = 31 AND MONTH_OF_DATE(dat) = 12;
	28:	(* 1st of january *)
		enabled := DAY_OF_YEAR(dat) = 1;
ELSE
	enabled := FALSE;
END_CASE;

(* set output if necessary *)
IF enabled AND NOT Q AND daytime >= start AND run_date <> dat THEN
	Q := TRUE;
	activation := tx;
	run_date := dat;
ELSIF Q AND tx - activation >= duration THEN
	Q := FALSE;
END_IF;
last_check := Tx;


(* revision history
hm 22.2.2007		rev 1.1
	changed VAR RETAIN PERSISTENT to VAR RETAIN for better compatibility
	wago lon contollers do not support persisitent

hm	15.9.2007		rev 1.2
	replaced Time() with T_PLC_MS for compatibility and performance reasons

hm	7. oct. 2008	rev 1.3
	changed function month to month_of_date

hm	20. oct. 2008	rev 1.4
	improved performance
	deleted unnecessary trunc

hm	22. dec. 2008	rev 1.5
	make sure timer_2 is executed in the first cycle

*)
END_FUNCTION_BLOCK

(* POU Time&Date/HOLIDAY, ST *)
FUNCTION_BLOCK HOLIDAY
VAR_INPUT
	DATE_IN : DATE;
	COUNTRY : INT;
	FRIDAY : BOOL;
	SATURDAY : BOOL;
	SUNDAY : BOOL;
END_VAR

VAR CONSTANT
	SIZE : INT := 29;
END_VAR
VAR_OUTPUT
	Y : BOOL;
	NAME : STRING(30);
END_VAR
VAR
	last_active : DATE;
	ostern: DATE;
	i: INT;
	jahr: INT;
	x_date: DATE;
	cx: INT;
	wdx: INT;
	check: HOLIDAY_DATA;
END_VAR

(*
version 1.6	21. oct. 2008
programmer 	hugo
tested by	tobias

holiday calculates if a given day is a holiday and displays the name of the holiday as string as well as a boolean flag to indicate a holiday.
the holidays are specified in the country setup under global constants.
a holiday can be of fixed date for example new years day on january 1st.
a holiday can have a fixed offset from easter sunday as for most church holidays.
a holiday can be a specific weekday before a fixed date, for example buss und bettag is the last wednesday before nov 23rd.
with a simple f_use flag any specific holiday can be turned on or off if needed.

*)
(* for performance reasons only activate once a day *)
IF last_active = date_in THEN RETURN; END_IF;

(* determine country *)
IF COUNTRY = 0 THEN
	cx := location.DEFAULT;
ELSE
	cx := MIN(location.LMAX, COUNTRY);
END_IF;

(* berechnung von ostern für das aktuelle jahr *)
jahr := YEAR_OF_DATE(date_in);
ostern := EASTER(jahr);
last_active := DATE_IN;
wdx := DAY_OF_WEEK(DATE_IN);

(* check array if today is holiday *)
Y := (wdx = 5 AND FRIDAY) OR (wdx = 6 AND SATURDAY) OR (wdx = 7 AND SUNDAY);
NAME := '';

FOR i := 0 TO size DO
	check := location.HOLIDAY[cx, i];
	x_date := SET_DATE(jahr, check.MONTH , check.DAY);
	IF check.USE = 1 AND check.MONTH > 0 THEN
		(* check for fixed date holiday *)
		IF x_date = date_in THEN
			Y := TRUE;
			NAME := check.NAME;
			RETURN;
		END_IF;
	ELSIF check.USE = 1 AND check.MONTH = 0 THEN
		(* check for holiday in reference to easter *)
		IF DATE_ADD(ostern, check.DAY ,0,0,0) = date_in THEN
			Y := TRUE;
			NAME := check.NAME;
			RETURN;
		END_IF;
	ELSIF check.USE < 0 THEN
		(* check for holiday on a weekday before date *)
		IF DAY_OF_WEEK(date_in) = ABS(check.USE) AND date_in < x_date AND date_in >= DATE_ADD(x_date,-7,0,0,0) THEN
			Y := TRUE;
			NAME := check.NAME;
			RETURN;
		END_IF;
	END_IF;
END_FOR;



(*
Neujahrstag 	1. Januar 	• 	• 	• 	• 	• 	• 	• 	• 	• 	• 	• 	• 	• 	• 	• 	•
Heilige Drei Könige 	6. Januar 	• 	• 												• 		
Karfreitag 	Ostersonntag - 2d 	• 	• 	• 	• 	• 	• 	• 	• 	• 	• 	• 	• 	• 	• 	• 	•
Ostersonntag 	siehe Osterdatum 				(•) 												
Ostermontag 	Ostersonntag + 1d 	• 	• 	• 	• 	• 	• 	• 	• 	• 	• 	• 	• 	• 	• 	• 	•
Tag der Arbeit 	1. Mai 	• 	• 	• 	• 	• 	• 	• 	• 	• 	• 	• 	• 	• 	• 	• 	•
Christi Himmelfahrt 	Ostersonntag + 39d 	• 	• 	• 	• 	• 	• 	• 	• 	• 	• 	• 	• 	• 	• 	• 	•
Pfingstsonntag 	Ostersonntag + 49d 				(•) 												
Pfingstmontag 	Ostersonntag + 50d 	• 	• 	• 	• 	• 	• 	• 	• 	• 	• 	• 	• 	• 	• 	• 	•
Fronleichnam 	Ostersonntag + 60d 	• 	• 					• 			• 	• 	• 	1) 			2)
Augsburger Friedensfest 	8. August 		(3) 														
Mariä Himmelfahrt 	15. August 		(5) 										• 				
Tag der Deutschen Einheit 	3. Oktober 6) 	• 	• 	• 	• 	• 	• 	• 	• 	• 	• 	• 	• 	• 	• 	• 	•
Reformationstag 	31. Oktober 				• 				• 					• 	• 		•
Allerheiligen 	1. November 	• 	• 								• 	• 	• 				
Buß- und Bettag 4) 	Mittwoch vor dem 23.11. 			7 										• 			
1. Weihnachtstag 	25. Dezember 	• 	• 	• 	• 	• 	• 	• 	• 	• 	• 	• 	• 	• 	• 	• 	•
2. Weihnachtstag 	26. Dezember 	• 	• 	• 	• 	• 	• 	• 	• 	• 	• 	• 	• 	• 	• 	• 	•
*)



(* revision history
hm 	27. feb. 2007	rev 1.1
	deleted unused variable init

hm	31. oct. 2007	rev 1.2
	changed holiday definition from constant to input constant to allow easier changes by user without recompilation of the lib

hm 	24. nov. 2007	rev 1.3
	changes F_use of  Buß_und_Bettag to 0 because this is no official holiday

hm	7. apr. 2008	rev 1.4
	improved performance

hm	7. oct. 2008	rev 1.5
	changed code to use setup data from global constants
	changed length of output NAME from 20 to 30
	holiday will now also be indicated on a weekend
	changed function year to year_of_date
	changed function weekday to day_of_week

hm	21. oct. 2008	rev 1.6
	using location constants
*)
END_FUNCTION_BLOCK

(* POU Time&Date/YEAR_OF_DATE, ST *)
FUNCTION YEAR_OF_DATE : INT
VAR_INPUT
	IDATE : DATE;
END_VAR


(*
version 1.4	7. oct. 2008
programmer 	hugo
tested by		oscat

returs the year of a date  
the function works for dates from 1970 - 2099 

*)
YEAR_OF_DATE := DWORD_TO_INT((DATE_TO_DWORD(idate)+43200) / 31557600 + 1970);


(* revision history
hm	4. aug 2006		rev 1.0
	original version

hm	1. okt 2007		rev 1.1
	corrected error in algorithm
	adjustment for S7 compatibility

hm	23.12.2007		rev 1.2
	changed code for better performance

hm	7. apr. 2008	rev 1.3
	deleted unused step7 code

hm	7. oct. 2008	rev 1.4
	reneamed function (year) to year_of_date

*)
END_FUNCTION

(* POU Time&Date/EASTER, ST *)
FUNCTION EASTER : DATE
VAR_INPUT
	year : INT;
END_VAR
VAR
	b,c: INT;
	oday: INT;
END_VAR

(*
version 1.3	7. apr. 2008
programmer 	hugo
tested by	tobias

easter calculates the day of easter sunday for a given year.
most other catholic holidays are calculated in reference to easter sunday.

*)
b := (204 - 11 * (YEAR MOD 19)) MOD 30;
IF b > 27 THEN b := b - 1; END_IF;
c := (year + SHR(year,2) + b - 13) MOD 7;
oday := 28 + b - c;
IF oday > 33 THEN
	easter := set_Date(year, 4, oday - 31);
ELSE
	EASTER := SET_DATE(year, 3, oday);
END_IF;




(* alternativer algorithmus ueber das pasah fest
execution time roughly 200us
Der sog. Passah-Vollmond wird berechnet, in dem das Jahr durch 19 ge-
teilt wird und der Rest mit der folgenden Tabelle verglichen wird:
 
    0: Apr 14       5: Apr 18      10: Mrz 25      15: Mrz 30
    1: Apr 03       6: Apr 08      11: Apr 13      16: Apr 17
    2: Mrz 23       7: Mrz 28      12: Apr 02      17: Apr 07
    3: Apr 11       8: Apr 16      13: Mrz 22      18: Mrz 27
    4: Mrz 31       9: Apr 05      14: Apr 10
 
Faellt dieses Datum auf einen Sonntag, ist Ostern der naechste Sonntag!
 
Beispiel: 1992 MOD 19 = 16, daraus folgt 17.04., der naechste Sonntag
          ist dann der 19. April (Ostersonntag)
*)


(* this algorithm is 180 us
a := year MOD 19;
b := year / 100;
c := year MOD 100;
d := b / 4;
e := b MOD 4;
f := (b + 8) / 25;
g := (b - f + 1) / 3;
h := (19 * a + b - d -g + 15) MOD 30;
i := C / 4;
k := c MOD 4;
l := (32 + 2*e + 2*i - h - k) MOD 7;
m := (a + 11 * h + 22 * l) / 451;
x := h + l - 7 * m + 114;
n := X / 31;
o := x MOD 31 + 1;

easter := set_Date(year,n,o);
*)
(*
Im Magazin "Nature" vom 20. April 1876 veröffentlichte ein anonymer Autor eine Tabelle mit Regeln zur Berechnung des (Gregorianischen) Ostersonntages des Jahres J. In Formeln ausgedrückt erhält man das Folgende:
a	=	J mod 19
b	=	int(J / 100)
c	=	J mod 100
d	=	int(b / 4)
e	=	b mod 4
f	=	int((b + 8) / 25)
g	=	int((b - f + 1) / 3
h	=	(19 · a + b - d - g + 15) mod 30
i	=	int(c / 4)
k	=	c mod 4
l	=	(32 + 2 · e + 2 · i - h - k) mod 7
m	=	int((a + 11 · h + 22 · l) / 451)
n	=	int((h + l - 7 · m + 114) / 31)
o	=	(h + l - 7 · m + 114) mod 31

n ist hierbei die Nummer des Monats, o + 1 die Nummer des Tages auf welchen der Ostersonntag im Jahr J fällt. Dieser Algorithmus kommt ohne Hilfszahlen aus.

*)

(* revision history
hm	27. dec 2006	rev 1.0
	original version

hm	15. dec 2007	rev 1.1
	modified code for better performance

hm	3. feb 2008		rev 1.2
	modified code for better performance

hm	7. apr. 2008	rev 1.3
	improved performance
*)
END_FUNCTION

(* POU Time&Date/SET_DATE, ST *)
FUNCTION SET_DATE : DATE
VAR_INPUT
	YEAR : INT;
	MONTH : INT;
	DAY : INT;
END_VAR
VAR
	count : DWORD;
END_VAR

(*
version 2.1	16. nov. 2008
programmer 	hugo
tested by	tobias

creates a date output from year, month and day of month   

*)
(* calculate the amount of days to 31.12. the year before *)
count := SHR(INT_TO_DWORD(year) * 1461 - 2878173,2)+INT_TO_DWORD(day);
(* add the days for the month of the year *)
count := count + INT_TO_DWORD(setup.MTH_OFS[LIMIT(1,month,12)]);
(* for leap years and month > february then add one more day *)
IF month > 2 AND LEAP_YEAR(year) THEN count := count + 1; END_IF;
(* generate the date *)
SET_DATE := DWORD_TO_DATE(count * 86400);



(* revision history
hm	4. aug. 2006	rev 1.0
	original version

hm	19 sep. 2007	rev 1.1
	use function leap_year to calculate leap year, more exceptions are handled

hm	1. okt	2007	rev 1.2
	added compatibility to step7

hm	16.dec 2007		rev 1.3
	changed code to improove performance

hm	3. jan. 2008	rev 1.4
	further improvements in performance

hm	16. mar. 2008	rev 1.5
	added type conversions to avoid warnings under codesys 3.0

hm	7. apr. 2008	rev 1.6
	deleted unused step7 code

hm	14. oct. 2008	rev 1.7
	optimized code for better performance

hm	25. oct. 2008	rev 2.0
	new code using setup constants

hm	16. nov. 2008	rev 2.1
	added typecats to avoid warnings
*)
END_FUNCTION

(* POU Time&Date/LEAP_YEAR, ST *)
FUNCTION LEAP_YEAR : BOOL
VAR_INPUT
	yr : INT;
END_VAR


(*
version 1.1	2 oct 2006
programmer 	hugo
tested by		tobias


leap_year is true if the tested year is a leap year  
  
*)
leap_year := SHL(yr,14) = 0;

(* this code was used prior to rev 1.1

IF yr MOD 400 = 0 THEN leap_year := TRUE;
ELSIF yr MOD 100 = 0 THEN leap_year := FALSE;
ELSIF yr MOD 4 =0 THEN leap_year := TRUE;
ELSE leap_year := FALSE;
END_IF;

*)

(* change history

hm 	2.10.2006		rev 1.1
	the function now works for any year from 1970 up to 2100

hm	1. oct 2007		rev 1.2
	chaged code for higher performance
*)
END_FUNCTION

(* POU Time&Date/DATE_ADD, ST *)
FUNCTION DATE_ADD : DATE
VAR_INPUT
	IDATE : DATE;
	D : INT;
	W : INT;
	M : INT;
	Y : INT;
END_VAR
VAR
	mo: INT;
	yr : INT;
END_VAR


(*
version 1.5	29. mar. 2009
programmer 	hugo
tested by		oscat

date_add adds days, weeks, month or years to a date.
negative inputs are allowed for subtraction.

*)
DATE_ADD := DWORD_TO_DATE(DATE_TO_DWORD(idate) + 86400 * INT_TO_DWORD(d) + 604800 * INT_TO_DWORD(w));
mo := MONTH_OF_DATE(DATE_ADD);
yr := YEAR_OF_DATE(DATE_ADD) + y + FLOOR(INT_TO_REAL(mo + m - 1) * 0.08333333333333);
mo := mo + (ABS(m) MOD 12) * SGN(m);
IF mo < 1 THEN
	mo := mo + 12;
ELSIF mo > 12 THEN
	mo := mo - 12;
END_IF;
DATE_ADD := SET_DATE(yr,mo,DAY_OF_MONTH(DATE_ADD));



(* revision history

hm 27.12.2006	rev 1.0
	nrw module

hm 12.4.2007		rev 1.1
	corrected an error while date would be incorrect when year  = 0

hm	1.11.2007		rev 1.2
	added int_to_dword stetements to avoid possible overrun with möller ecp4

hm	22. mar. 2008	rev 1.3
	fixed some bugs when month was negative

hm	7. oct. 2008	rev 1.4
	changed function year to year_of_date
	changed function month to month_of_date

hm	29. mar. 2009	rev 1.5
	improved performance
*)
END_FUNCTION

(* POU Time&Date/MONTH_OF_DATE, ST *)
FUNCTION MONTH_OF_DATE : INT
VAR_INPUT
	IDATE : DATE;
END_VAR


(*
version 1.3	27. mar. 2009
programmer 	hugo
tested by		tobias

returns the current month of the year.

*)
MONTH_OF_DATE := DAY_OF_YEAR(idate);
IF MONTH_OF_DATE < 32 THEN
	MONTH_OF_DATE := 1;
ELSIF LEAP_OF_DATE(IDATE) THEN
	MONTH_OF_DATE := (MONTH_OF_DATE * 53 + 1668) / 1623;
ELSE
	MONTH_OF_DATE := (MONTH_OF_DATE * 53 + 1700) / 1620;
END_IF;


(* code for rev 1.2
MONTH_OF_DATE := DAY_OF_YEAR(IDATE);
IF LEAP_OF_DATE(IDATE) THEN
	CASE MONTH_OF_DATE OF
		1..31 	:	MONTH_OF_DATE := 1;
		32..60	:	MONTH_OF_DATE := 2;
		61..91	:	MONTH_OF_DATE := 3;
		92..121 :	MONTH_OF_DATE := 4;
		122..152:	MONTH_OF_DATE := 5;
		153..182:	MONTH_OF_DATE := 6;
		183..213:	MONTH_OF_DATE := 7;
		214..244:	MONTH_OF_DATE := 8;
		245..274:	MONTH_OF_DATE := 9;
		275..305:	MONTH_OF_DATE := 10;
		306..335:	MONTH_OF_DATE := 11;
		336..366:	MONTH_OF_DATE := 12;
	END_CASE;
ELSE
	CASE MONTH_OF_DATE OF
		1..31 	:	MONTH_OF_DATE := 1;
		32..59	:	MONTH_OF_DATE := 2;
		60..90	:	MONTH_OF_DATE := 3;
		91..120 :	MONTH_OF_DATE := 4;
		121..151:	MONTH_OF_DATE := 5;
		152..181:	MONTH_OF_DATE := 6;
		182..212:	MONTH_OF_DATE := 7;
		213..243:	MONTH_OF_DATE := 8;
		244..273:	MONTH_OF_DATE := 9;
		274..304:	MONTH_OF_DATE := 10;
		305..334:	MONTH_OF_DATE := 11;
		335..365:	MONTH_OF_DATE := 12;
	END_CASE;
END_IF;
*)


(* revision history
hm	1. aug 2006	rev 1.0
	original version	

hm	1. okt 2007	rev 1.1
	replaced old code (string conversion) with mathematics
	the execution time is now multiple times faster.

hm	7. oct. 2008	rev 1.2
	changed name of function from month to MONTH_OF_DATE

hm	27. mar. 2009	rev 1.3
	new improved code

*)
END_FUNCTION

(* POU Time&Date/DAY_OF_YEAR, ST *)
FUNCTION DAY_OF_YEAR : INT
VAR_INPUT
	IDATE : DATE;
END_VAR


(*
version 1.3	7. oct. 2008
programmer 	hugo
tested by	oscat

calculates the day of the year

*)
DAY_OF_YEAR := DWORD_TO_INT((DATE_TO_DWORD(idate) - DATE_TO_DWORD(YEAR_BEGIN(YEAR_OF_DATE(idate)))) / 86400) + 1;



(* revivision history
hm	4. aug. 2007		rev 1.0
	original version

hm	1. oct. 2007		rev 1.1
	added compatibility to STEP7

hm	4. jan. 2008		rev 1.2
	changed code for better performance

hm	7. oct. 2008		rev 1.3
	changed name of function year to year_of_date

*)
END_FUNCTION

(* POU Time&Date/YEAR_BEGIN, ST *)
FUNCTION YEAR_BEGIN : DATE
VAR_INPUT
	y : INT;
END_VAR


(*
version 1.2	7. Apr. 2008
programmer 	hugo
tested by	tobias

returs the date of january 1st for the given year  
the function works for dates from 1970 - 2099 

*)
YEAR_BEGIN := DWORD_TO_DATE(SHR(INT_TO_DWORD(y) * 1461 - 2878169,2)*86400);



(* revision history
hm	19. dec 2007	rev 1.0
	original version

hm	4. jan 2008		rev 1.1
	formula for step7 was incorrect during leap years

hm	7. apr. 2008	rev 1.2
	deleted unused step7 code
*)
END_FUNCTION

(* POU Time&Date/LEAP_OF_DATE, ST *)
FUNCTION LEAP_OF_DATE : BOOL
VAR_INPUT
	idate : DATE;
END_VAR


(*
version 1.2	8 jan 2008
programmer 	hugo
tested by		tobias

leap_year is true if the tested year is a leap year  

*)
leap_of_Date := SHL(DWORD_TO_INT((DATE_TO_DWORD(idate)+43200) / 31557600)+2,14) = 0;


(* change history

2.10.2006		rev 1.1
the function now calls leap_year to accomodate further accuracy.
the function now works for any year from 1970 to 2100

8. jan 2008		rev 1.2
	improved code for better performance
*)
END_FUNCTION

(* POU Mathematical/FLOOR, ST *)
FUNCTION FLOOR : INT
VAR_INPUT
	X : REAL;
END_VAR


(*
version 1.1	21. mar. 2008
programmer 	hugo
tested by		tobias

This is a rounding function which returns the biggest possible integer which is less or equal to X.
floor(3.14) = 3
floor(-3.14) = -4

*)
FLOOR := REAL_TO_INT(X);
IF FLOOR > X THEN
	FLOOR := FLOOR - 1;
END_IF;

(* revision history
hm		7. feb 2007		rev 1.0
	originlal version

hm		21. mar. 2008	rev 1.1
	replaced trunc with real_to_int for compatibility reasons

*)
END_FUNCTION

(* POU Mathematical/SGN, ST *)
FUNCTION SGN : INT
VAR_INPUT
	X : REAL;
END_VAR


(*
version 1.1	11. nov. 2008
programmer 	hugo
tested by	tobias

sgn returns 0 when X = 0 , -1 when X < 1 and +1 when X > 1

*)
IF X > 0 THEN
	SGN := 1;
ELSIF X < 0 THEN
	SGN := -1;
ELSE
	SGN := 0;
END_IF;



(* revision histroy
hm	16. oct 2007	rev 1.0
	original version

hm	11. nov 2007	rev 1.1
	changed type of function from real to int

*)
END_FUNCTION

(* POU Time&Date/DAY_OF_MONTH, ST *)
FUNCTION DAY_OF_MONTH : INT
VAR_INPUT
	IDATE : DATE;
END_VAR
VAR
	leap: INT;
END_VAR

(*
version 2.1	10. mar. 2009
programmer 	hugo
tested by		tobias

returns the day OF month for any DATE

*)
(* calculate the day in the year *)
DAY_OF_MONTH := DAY_OF_YEAR(idate);
(* leap will be set to one for a leap year *)
leap := BOOL_TO_INT(LEAP_OF_DATE(idate));
(* if leap year deduct one from the days of the year *)
DAY_OF_MONTH := DAY_OF_MONTH - leap;
(* search if we are in month december to march ? *)
IF DAY_OF_MONTH > setup.MTH_OFS[9] THEN
	IF DAY_OF_MONTH > setup.MTH_OFS[11] THEN
		IF DAY_OF_MONTH > setup.mth_ofs[12] THEN
			DAY_OF_MONTH := DAY_OF_MONTH - setup.MTH_OFS[12];
		ELSE
			DAY_OF_MONTH := DAY_OF_MONTH - setup.MTH_OFS[11];
		END_IF;
	ELSE
		IF DAY_OF_MONTH > setup.mth_ofs[10] THEN
			DAY_OF_MONTH := DAY_OF_MONTH - setup.MTH_OFS[10];
		ELSE
			DAY_OF_MONTH := DAY_OF_MONTH - setup.MTH_OFS[9];
		END_IF;
	END_IF;
ELSIF DAY_OF_MONTH > setup.MTH_OFS[5] THEN
	IF DAY_OF_MONTH > setup.MTH_OFS[7] THEN
		IF DAY_OF_MONTH > setup.mth_ofs[8] THEN
			DAY_OF_MONTH := DAY_OF_MONTH - setup.MTH_OFS[8];
		ELSE
			DAY_OF_MONTH := DAY_OF_MONTH - setup.MTH_OFS[7];
		END_IF;
	ELSE
		IF DAY_OF_MONTH > setup.mth_ofs[6] THEN
			DAY_OF_MONTH := DAY_OF_MONTH - setup.MTH_OFS[6];
		ELSE
			DAY_OF_MONTH := DAY_OF_MONTH - setup.MTH_OFS[5];
		END_IF;
	END_IF;
ELSIF DAY_OF_MONTH > setup.MTH_OFS[3] THEN
	IF DAY_OF_MONTH > setup.MTH_OFS[4] THEN
		DAY_OF_MONTH := DAY_OF_MONTH - setup.MTH_OFS[4];
	ELSE
		DAY_OF_MONTH := DAY_OF_MONTH - setup.MTH_OFS[3];
	END_IF;
ELSE
	(* since now we must be in february or january we need to add leap again *)
	DAY_OF_MONTH := DAY_OF_MONTH + leap;
	IF DAY_OF_MONTH > setup.MTH_OFS[2] THEN DAY_OF_MONTH := DAY_OF_MONTH - setup.mth_ofs[2]; END_IF;
	(* since nothing was true before, day_of_month must already be good *)
END_IF;


(*
Revision history

hm 22.1.2007		rev 1.1
	deleted unused variable day_in_year and day_in_year_begin

hm	1. okt 2007	rev 1.2
	changed code to use day_of_year and leap_of_date
	added compatibility to STEP7

hm	8. oct 2007	rev 1.3
	deleted unused variable yr

hm	8. jan 2008	rev 1.4
	improved performance

hm	25. oct. 2008	rev 2.0
	new code using setup constants

